C03654=1204.977,411.495,-82.961,-175.836,8.473,148.470
C03655=1204.981,411.248,-82.925,-175.837,8.471,148.469
C03656=1204.985,411.000,-82.891,-175.837,8.469,148.469
C03657=1204.989,410.753,-82.855,-175.837,8.467,148.468
C03658=1204.993,410.506,-82.820,-175.838,8.464,148.468
C03659=1204.997,410.258,-82.785,-175.838,8.462,148.467
C03660=1205.001,410.011,-82.749,-175.839,8.460,148.467
C03661=1205.005,409.764,-82.714,-175.839,8.458,148.466
C03662=1205.009,409.516,-82.679,-175.839,8.456,148.466
C03663=1205.013,409.268,-82.644,-175.839,8.453,148.465
C03664=1205.017,409.021,-82.609,-175.840,8.451,148.465
C03665=1205.021,408.773,-82.574,-175.840,8.449,148.464
C03666=1205.025,408.525,-82.539,-175.840,8.447,148.464
C03667=1205.029,408.278,-82.504,-175.840,8.445,148.463
C03668=1205.032,408.031,-82.469,-175.841,8.443,148.463
C03669=1205.037,407.784,-82.434,-175.841,8.440,148.462
C03670=1205.040,407.536,-82.399,-175.842,8.438,148.462
C03671=1205.044,407.288,-82.364,-175.842,8.436,148.461
C03672=1205.049,407.041,-82.329,-175.842,8.433,148.461
C03673=1205.053,406.793,-82.294,-175.843,8.431,148.460
C03674=1205.057,406.546,-82.259,-175.843,8.428,148.460
C03675=1205.061,406.298,-82.224,-175.844,8.426,148.459
C03676=1205.065,406.051,-82.188,-175.844,8.424,148.459
C03677=1205.069,405.803,-82.154,-175.844,8.422,148.458
C03678=1205.073,405.556,-82.118,-175.845,8.420,148.458
C03679=1205.077,405.308,-82.084,-175.845,8.417,148.457
C03680=1205.081,405.061,-82.048,-175.845,8.415,148.457
C03681=1205.085,404.813,-82.014,-175.846,8.412,148.456
C03682=1205.089,404.566,-81.978,-175.847,8.410,148.456
C03683=1205.093,404.318,-81.944,-175.847,8.408,148.455
C03684=1205.098,404.071,-81.908,-175.847,8.405,148.455
C03685=1205.101,403.823,-81.874,-175.847,8.403,148.454
C03686=1205.104,403.576,-81.839,-175.848,8.401,148.454
C03687=1205.109,403.328,-81.804,-175.849,8.398,148.453
C03688=1205.113,403.081,-81.769,-175.849,8.396,148.453
C03689=1205.117,402.833,-81.734,-175.849,8.394,148.452
C03690=1205.121,402.586,-81.699,-175.849,8.391,148.452
C03691=1205.125,402.338,-81.664,-175.850,8.389,148.451
C03692=1205.129,402.090,-81.629,-175.851,8.386,148.451
C03693=1205.133,401.843,-81.594,-175.851,8.384,148.450
C03694=1205.138,401.595,-81.559,-175.851,8.382,148.450
C03695=1205.141,401.348,-81.524,-175.852,8.379,148.449
C03696=1205.145,401.101,-81.490,-175.852,8.376,148.449
C03697=1205.149,400.853,-81.455,-175.853,8.374,148.448
C03698=1205.153,400.606,-81.420,-175.853,8.372,148.448
C03699=1205.157,400.358,-81.385,-175.853,8.370,148.447
C03700=1205.162,400.111,-81.350,-175.854,8.367,148.447
C03701=1205.166,399.863,-81.315,-175.854,8.364,148.446
C03702=1205.170,399.615,-81.280,-175.855,8.362,148.446
C03703=1205.173,399.368,-81.246,-175.856,8.359,148.445
C03704=1205.177,399.120,-81.211,-175.856,8.357,148.445
C03705=1205.182,398.873,-81.176,-175.856,8.355,148.444
C03706=1205.185,398.625,-81.141,-175.857,8.352,148.444
C03707=1205.190,398.378,-81.106,-175.858,8.350,148.443
C03708=1205.194,398.130,-81.071,-175.858,8.347,148.443
C03709=1205.197,397.883,-81.037,-175.859,8.344,148.442
C03710=1205.201,397.635,-81.002,-175.859,8.342,148.442
C03711=1205.206,397.388,-80.968,-175.860,8.340,148.441
C03712=1205.210,397.140,-80.932,-175.860,8.337,148.441
C03713=1205.214,396.893,-80.898,-175.861,8.335,148.440
C03714=1205.218,396.645,-80.863,-175.861,8.332,148.440
C03715=1205.222,396.398,-80.828,-175.862,8.329,148.439
C03716=1205.226,396.150,-80.793,-175.862,8.327,148.439
C03717=1205.230,395.903,-80.759,-175.863,8.324,148.438
C03718=1205.234,395.654,-80.724,-175.863,8.322,148.438
C03719=1205.238,395.408,-80.689,-175.864,8.319,148.437
C03720=1205.242,395.160,-80.655,-175.865,8.317,148.437
C03721=1205.246,394.912,-80.620,-175.865,8.314,148.436
C03722=1205.250,394.664,-80.585,-175.866,8.312,148.436
C03723=1205.254,394.417,-80.550,-175.866,8.309,148.435
C03724=1205.258,394.170,-80.516,-175.867,8.307,148.435
C03725=1205.262,393.922,-80.481,-175.868,8.303,148.434
C03726=1205.266,393.674,-80.447,-175.868,8.301,148.433
C03727=1205.270,393.427,-80.411,-175.869,8.298,148.433
C03728=1205.274,393.180,-80.377,-175.869,8.296,148.433
C03729=1205.279,392.896,-80.337,-175.870,8.293,148.432
C03730=1205.283,392.614,-80.298,-175.871,8.290,148.431
C03731=1205.288,392.332,-80.259,-175.872,8.287,148.431
C03732=1205.293,392.049,-80.219,-175.873,8.284,148.430
C03733=1205.297,391.801,-80.184,-175.873,8.281,148.430
C03734=1205.301,391.554,-80.150,-175.873,8.278,148.429
C03735=1205.305,391.306,-80.115,-175.874,8.276,148.429
C03736=1205.309,391.059,-80.080,-175.875,8.273,148.428
C03737=1205.312,390.811,-80.046,-175.876,8.270,148.428
C03738=1205.317,390.564,-80.012,-175.876,8.268,148.427
C03739=1205.321,390.316,-79.977,-175.877,8.265,148.427
C03740=1205.325,390.068,-79.942,-175.877,8.263,148.426
C03741=1205.328,389.821,-79.908,-175.879,8.260,148.426
C03742=1205.333,389.573,-79.874,-175.879,8.257,148.425
C03743=1205.337,389.326,-79.839,-175.880,8.255,148.425
C03744=1205.341,389.078,-79.805,-175.881,8.252,148.424
C03745=1205.345,388.830,-79.770,-175.881,8.249,148.424
C03746=1205.349,388.583,-79.735,-175.882,8.246,148.423
C03747=1205.353,388.336,-79.701,-175.883,8.244,148.423
C03748=1205.357,388.088,-79.666,-175.884,8.240,148.422
C03749=1205.361,387.840,-79.632,-175.884,8.238,148.422
C03750=1205.365,387.593,-79.598,-175.885,8.235,148.421
C03751=1205.369,387.345,-79.563,-175.886,8.232,148.421
C03752=1205.374,387.098,-79.529,-175.887,8.229,148.420
C03753=1205.377,386.850,-79.494,-175.887,8.227,148.420
C03754=1205.381,386.602,-79.460,-175.888,8.224,148.419
C03755=1205.385,386.355,-79.426,-175.889,8.221,148.419
C03756=1205.389,386.107,-79.391,-175.890,8.218,148.418
C03757=1205.394,385.860,-79.357,-175.891,8.215,148.418
C03758=1205.397,385.612,-79.322,-175.891,8.213,148.417
C03759=1205.402,385.365,-79.288,-175.893,8.210,148.417
C03760=1205.406,385.116,-79.253,-175.893,8.207,148.416
C03761=1205.409,384.869,-79.219,-175.894,8.204,148.416
C03762=1205.414,384.622,-79.185,-175.895,8.201,148.415
C03763=1205.417,384.374,-79.151,-175.896,8.199,148.415
C03764=1205.422,384.127,-79.116,-175.897,8.196,148.414
C03765=1205.425,383.879,-79.082,-175.898,8.193,148.414
C03766=1205.430,383.631,-79.048,-175.899,8.190,148.413
C03767=1205.434,383.383,-79.014,-175.900,8.187,148.413
C03768=1205.438,383.136,-78.979,-175.901,8.184,148.412
C03769=1205.442,382.888,-78.945,-175.902,8.181,148.412
C03770=1205.446,382.641,-78.911,-175.903,8.178,148.411
C03771=1205.450,382.393,-78.876,-175.903,8.176,148.411
C03772=1205.454,382.146,-78.842,-175.904,8.173,148.410
C03773=1205.458,381.898,-78.808,-175.905,8.171,148.410
C03774=1205.462,381.650,-78.774,-175.906,8.167,148.409
C03775=1205.467,381.403,-78.740,-175.907,8.165,148.409
C03776=1205.471,381.154,-78.705,-175.908,8.162,148.408
C03777=1205.474,380.907,-78.671,-175.909,8.159,148.408
C03778=1205.479,380.660,-78.637,-175.911,8.156,148.408
C03779=1205.482,380.412,-78.603,-175.911,8.153,148.407
C03780=1205.487,380.164,-78.569,-175.913,8.150,148.407
C03781=1205.491,379.917,-78.535,-175.913,8.147,148.406
C03782=1205.495,379.669,-78.500,-175.915,8.144,148.406
C03783=1205.499,379.422,-78.466,-175.916,8.141,148.405
C03784=1205.503,379.174,-78.432,-175.916,8.138,148.405
C03785=1205.507,378.926,-78.398,-175.918,8.135,148.404
C03786=1205.511,378.678,-78.364,-175.919,8.133,148.404
C03787=1205.515,378.431,-78.330,-175.920,8.129,148.403
C03788=1205.518,378.184,-78.296,-175.921,8.127,148.403
C03789=1205.523,377.936,-78.262,-175.922,8.124,148.402
C03790=1205.527,377.688,-78.228,-175.923,8.121,148.402
C03791=1205.532,377.441,-78.194,-175.924,8.118,148.401
C03792=1205.535,377.193,-78.160,-175.926,8.114,148.401
C03793=1205.540,376.945,-78.126,-175.927,8.111,148.401
C03794=1205.544,376.698,-78.092,-175.928,8.108,148.400
C03795=1205.547,376.450,-78.058,-175.929,8.106,148.400
C03796=1205.552,376.202,-78.024,-175.930,8.103,148.399
C03797=1205.556,375.955,-77.990,-175.931,8.100,148.399
C03798=1205.560,375.707,-77.956,-175.933,8.097,148.398
C03799=1205.564,375.459,-77.922,-175.933,8.094,148.398
C03800=1205.568,375.212,-77.888,-175.935,8.090,148.397
C03801=1205.572,374.964,-77.854,-175.936,8.088,148.397
C03802=1205.576,374.716,-77.820,-175.938,8.085,148.397
C03803=1205.581,374.468,-77.786,-175.939,8.082,148.396
C03804=1205.584,374.221,-77.752,-175.940,8.079,148.396
C03805=1205.588,373.974,-77.718,-175.941,8.076,148.396
C03806=1205.592,373.725,-77.684,-175.943,8.072,148.395
C03807=1205.596,373.478,-77.650,-175.944,8.070,148.394
C03808=1205.600,373.230,-77.617,-175.945,8.067,148.394
C03809=1205.605,372.983,-77.583,-175.946,8.064,148.394
C03810=1205.609,372.735,-77.549,-175.947,8.061,148.393
C03811=1205.612,372.487,-77.515,-175.949,8.058,148.393
C03812=1205.617,372.239,-77.482,-175.950,8.055,148.392
C03813=1205.621,371.992,-77.448,-175.952,8.052,148.392
C03814=1205.625,371.744,-77.414,-175.953,8.049,148.392
C03815=1205.629,371.496,-77.380,-175.955,8.045,148.391
C03816=1205.633,371.249,-77.347,-175.956,8.043,148.391
C03817=1205.637,371.002,-77.313,-175.957,8.040,148.390
C03818=1205.641,370.754,-77.280,-175.958,8.037,148.390
C03819=1205.645,370.506,-77.245,-175.960,8.033,148.390
C03820=1205.649,370.258,-77.212,-175.961,8.031,148.389
C03821=1205.653,370.011,-77.178,-175.962,8.028,148.389
C03822=1205.657,369.763,-77.145,-175.964,8.024,148.388
C03823=1205.662,369.515,-77.111,-175.965,8.021,148.388
C03824=1205.665,369.267,-77.077,-175.966,8.019,148.388
C03825=1205.670,369.020,-77.044,-175.968,8.015,148.387
C03826=1205.673,368.773,-77.010,-175.970,8.012,148.387
C03827=1205.678,368.524,-76.976,-175.971,8.010,148.387
C03828=1205.682,368.277,-76.943,-175.973,8.006,148.386
C03829=1205.686,368.030,-76.909,-175.974,8.003,148.386
C03830=1205.690,367.781,-76.875,-175.975,8.000,148.385
C03831=1205.695,367.533,-76.842,-175.977,7.997,148.385
C03832=1205.699,367.286,-76.808,-175.978,7.994,148.385
C03833=1205.703,367.005,-76.771,-175.980,7.990,148.384
C03834=1205.708,366.725,-76.732,-175.982,7.987,148.384
C03835=1205.712,366.445,-76.695,-175.983,7.984,148.383
C03836=1205.717,366.164,-76.656,-175.985,7.980,148.383
C03837=1205.721,365.917,-76.623,-175.987,7.977,148.383
C03838=1205.725,365.669,-76.590,-175.988,7.974,148.382
C03839=1205.729,365.421,-76.557,-175.990,7.971,148.382
C03840=1205.733,365.173,-76.522,-175.992,7.968,148.382
C03841=1205.737,364.925,-76.489,-175.993,7.965,148.381
C03842=1205.742,364.678,-76.455,-175.995,7.961,148.381
C03843=1205.746,364.430,-76.422,-175.996,7.959,148.381
C03844=1205.750,364.182,-76.389,-175.998,7.955,148.380
C03845=1205.754,363.935,-76.355,-175.999,7.952,148.380
C03846=1205.758,363.687,-76.322,-176.001,7.949,148.380
C03847=1205.762,363.440,-76.289,-176.003,7.946,148.379
C03848=1205.766,363.191,-76.255,-176.004,7.944,148.379
C03849=1205.770,362.943,-76.222,-176.006,7.940,148.379
C03850=1205.774,362.696,-76.189,-176.007,7.937,148.378
C03851=1205.778,362.448,-76.156,-176.009,7.934,148.378
C03852=1205.782,362.200,-76.123,-176.011,7.931,148.378
C03853=1205.787,361.953,-76.088,-176.012,7.927,148.377
C03854=1205.791,361.705,-76.055,-176.014,7.925,148.377
C03855=1205.795,361.457,-76.022,-176.016,7.921,148.376
C03856=1205.799,361.210,-75.989,-176.018,7.919,148.376
C03857=1205.803,360.962,-75.956,-176.019,7.915,148.376
C03858=1205.807,360.714,-75.923,-176.021,7.913,148.376
C03859=1205.811,360.466,-75.889,-176.023,7.909,148.375
C03860=1205.816,360.219,-75.856,-176.024,7.906,148.375
C03861=1205.820,359.971,-75.823,-176.026,7.903,148.375
C03862=1205.823,359.723,-75.790,-176.028,7.900,148.374
C03863=1205.827,359.475,-75.756,-176.030,7.897,148.374
C03864=1205.832,359.227,-75.723,-176.031,7.894,148.374
C03865=1205.836,358.979,-75.690,-176.033,7.891,148.373
C03866=1205.839,358.732,-75.658,-176.035,7.888,148.373
C03867=1205.843,358.484,-75.624,-176.036,7.884,148.373
C03868=1205.847,358.236,-75.591,-176.038,7.882,148.373
C03869=1205.852,357.989,-75.558,-176.040,7.879,148.372
C03870=1205.856,357.740,-75.526,-176.042,7.875,148.372
C03871=1205.860,357.493,-75.492,-176.044,7.872,148.372
C03872=1205.864,357.245,-75.459,-176.046,7.869,148.371
C03873=1205.868,356.997,-75.426,-176.047,7.866,148.371
C03874=1205.873,356.749,-75.393,-176.049,7.863,148.371
C03875=1205.877,356.502,-75.360,-176.050,7.860,148.370
C03876=1205.881,356.254,-75.327,-176.053,7.857,148.370
C03877=1205.885,356.006,-75.294,-176.054,7.854,148.370
C03878=1205.889,355.758,-75.262,-176.056,7.851,148.370
C03879=1205.893,355.510,-75.229,-176.058,7.848,148.369
C03880=1205.897,355.263,-75.195,-176.060,7.845,148.369
C03881=1205.901,355.015,-75.162,-176.062,7.841,148.369
C03882=1205.906,354.767,-75.130,-176.063,7.839,148.369
C03883=1205.910,354.520,-75.097,-176.066,7.835,148.368
C03884=1205.914,354.272,-75.064,-176.067,7.833,148.368
C03885=1205.918,354.025,-75.031,-176.069,7.829,148.368
C03886=1205.922,353.776,-74.999,-176.071,7.827,148.368
C03887=1205.926,353.528,-74.966,-176.073,7.823,148.367
C03888=1205.930,353.281,-74.933,-176.075,7.820,148.367
C03889=1205.935,353.033,-74.899,-176.076,7.817,148.367
C03890=1205.938,352.785,-74.868,-176.079,7.814,148.366
C03891=1205.942,352.537,-74.834,-176.080,7.811,148.366
C03892=1205.947,352.289,-74.801,-176.082,7.808,148.366
C03893=1205.951,352.041,-74.769,-176.084,7.805,148.366
C03894=1205.955,351.793,-74.736,-176.086,7.802,148.365
C03895=1205.959,351.545,-74.704,-176.088,7.798,148.365
C03896=1205.964,351.298,-74.671,-176.090,7.796,148.365
C03897=1205.968,351.051,-74.638,-176.092,7.792,148.365
C03898=1205.972,350.802,-74.605,-176.094,7.790,148.365
C03899=1205.976,350.555,-74.573,-176.096,7.787,148.364
C03900=1205.980,350.306,-74.540,-176.097,7.784,148.364
C03901=1205.984,350.059,-74.507,-176.099,7.780,148.364
C03902=1205.988,349.811,-74.475,-176.101,7.777,148.364
C03903=1205.992,349.563,-74.442,-176.103,7.775,148.363
C03904=1205.997,349.315,-74.410,-176.105,7.771,148.363
C03905=1206.001,349.068,-74.377,-176.107,7.769,148.363
C03906=1206.005,348.820,-74.345,-176.109,7.765,148.363
C03907=1206.009,348.572,-74.312,-176.111,7.762,148.363
C03908=1206.014,348.323,-74.280,-176.113,7.760,148.362
C03909=1206.017,348.076,-74.247,-176.115,7.756,148.362
C03910=1206.022,347.828,-74.215,-176.117,7.754,148.362
C03911=1206.026,347.581,-74.182,-176.119,7.750,148.362
C03912=1206.030,347.333,-74.150,-176.121,7.747,148.362
C03913=1206.034,347.085,-74.117,-176.123,7.745,148.361
C03914=1206.038,346.837,-74.085,-176.125,7.741,148.361
C03915=1206.042,346.589,-74.052,-176.127,7.739,148.361
C03916=1206.047,346.342,-74.020,-176.129,7.735,148.361
C03917=1206.051,346.093,-73.988,-176.131,7.732,148.360
C03918=1206.055,345.846,-73.955,-176.133,7.729,148.360
C03919=1206.058,345.598,-73.923,-176.135,7.726,148.360
C03920=1206.063,345.349,-73.890,-176.137,7.724,148.360
C03921=1206.068,345.102,-73.858,-176.139,7.720,148.360
C03922=1206.071,344.854,-73.826,-176.141,7.717,148.359
C03923=1206.076,344.606,-73.793,-176.143,7.714,148.359
C03924=1206.079,344.358,-73.761,-176.145,7.711,148.359
C03925=1206.084,344.111,-73.729,-176.147,7.709,148.359
C03926=1206.088,343.863,-73.697,-176.149,7.705,148.359
C03927=1206.092,343.614,-73.664,-176.151,7.702,148.358
C03928=1206.096,343.366,-73.633,-176.153,7.699,148.358
C03929=1206.101,343.119,-73.600,-176.155,7.696,148.358
C03930=1206.104,342.871,-73.568,-176.157,7.694,148.358
C03931=1206.109,342.623,-73.535,-176.159,7.690,148.358
C03932=1206.113,342.375,-73.504,-176.162,7.687,148.358
C03933=1206.118,342.127,-73.472,-176.163,7.685,148.357
C03934=1206.121,341.880,-73.439,-176.166,7.681,148.357
C03935=1206.125,341.632,-73.407,-176.167,7.679,148.357
C03936=1206.129,341.384,-73.375,-176.169,7.675,148.357
C03937=1206.134,341.106,-73.338,-176.172,7.672,148.357
C03938=1206.140,340.827,-73.303,-176.174,7.669,148.357
C03939=1206.144,340.549,-73.266,-176.177,7.666,148.356
C03940=1206.148,340.271,-73.231,-176.179,7.662,148.356
C03941=1206.153,340.023,-73.198,-176.181,7.659,148.356
C03942=1206.157,339.775,-73.167,-176.183,7.657,148.356
C03943=1206.162,339.527,-73.134,-176.185,7.653,148.356
C03944=1206.165,339.279,-73.103,-176.188,7.650,148.356
C03945=1206.169,339.031,-73.071,-176.189,7.648,148.355
C03946=1206.174,338.783,-73.039,-176.191,7.644,148.355
C03947=1206.178,338.535,-73.007,-176.194,7.641,148.355
C03948=1206.181,338.287,-72.975,-176.196,7.639,148.355
C03949=1206.187,338.040,-72.943,-176.198,7.635,148.355
C03950=1206.190,337.792,-72.911,-176.200,7.633,148.355
C03951=1206.194,337.544,-72.879,-176.202,7.630,148.354
C03952=1206.199,337.296,-72.847,-176.204,7.627,148.354
C03953=1206.203,337.048,-72.815,-176.206,7.624,148.354
C03954=1206.206,336.800,-72.783,-176.208,7.621,148.354
C03955=1206.211,336.552,-72.751,-176.211,7.618,148.354
C03956=1206.215,336.304,-72.720,-176.213,7.615,148.354
C03957=1206.219,336.057,-72.688,-176.215,7.612,148.354
C03958=1206.224,335.808,-72.656,-176.217,7.609,148.353
C03959=1206.228,335.560,-72.625,-176.219,7.606,148.353
C03960=1206.232,335.312,-72.593,-176.221,7.603,148.353
C03961=1206.236,335.064,-72.561,-176.223,7.600,148.353
C03962=1206.240,334.816,-72.529,-176.226,7.597,148.353
C03963=1206.245,334.569,-72.497,-176.228,7.594,148.353
C03964=1206.248,334.321,-72.465,-176.230,7.591,148.353
C03965=1206.253,334.073,-72.435,-176.232,7.588,148.353
C03966=1206.257,333.824,-72.402,-176.234,7.586,148.352
C03967=1206.261,333.576,-72.370,-176.236,7.583,148.352
C03968=1206.265,333.329,-72.339,-176.239,7.580,148.352
C03969=1206.269,333.081,-72.307,-176.241,7.577,148.352
C03970=1206.274,332.833,-72.276,-176.243,7.574,148.352
C03971=1206.278,332.585,-72.244,-176.245,7.571,148.352
C03972=1206.283,332.337,-72.212,-176.247,7.568,148.352
C03973=1206.287,332.089,-72.181,-176.250,7.565,148.352
C03974=1206.291,331.841,-72.150,-176.251,7.563,148.351
C03975=1206.295,331.593,-72.118,-176.254,7.560,148.351
C03976=1206.299,331.344,-72.086,-176.256,7.556,148.351
C03977=1206.304,331.097,-72.055,-176.258,7.554,148.351
C03978=1206.307,330.849,-72.023,-176.261,7.551,148.351
C03979=1206.312,330.601,-71.992,-176.263,7.547,148.351
C03980=1206.316,330.353,-71.960,-176.265,7.545,148.351
C03981=1206.320,330.106,-71.929,-176.267,7.542,148.351
C03982=1206.324,329.857,-71.898,-176.269,7.540,148.351
C03983=1206.328,329.610,-71.866,-176.272,7.536,148.350
C03984=1206.332,329.361,-71.835,-176.274,7.533,148.350
C03985=1206.337,329.113,-71.803,-176.276,7.531,148.350
C03986=1206.341,328.865,-71.772,-176.279,7.528,148.350
C03987=1206.346,328.617,-71.740,-176.281,7.524,148.350
C03988=1206.349,328.369,-71.709,-176.283,7.522,148.350
C03989=1206.354,328.121,-71.678,-176.285,7.519,148.350
C03990=1206.358,327.873,-71.646,-176.287,7.517,148.350
C03991=1206.362,327.625,-71.615,-176.289,7.513,148.350
C03992=1206.366,327.377,-71.583,-176.292,7.510,148.350
C03993=1206.371,327.129,-71.553,-176.294,7.508,148.350
C03994=1206.375,326.881,-71.522,-176.296,7.505,148.350
C03995=1206.379,326.633,-71.490,-176.299,7.501,148.349
C03996=1206.384,326.385,-71.459,-176.301,7.499,148.349
C03997=1206.387,326.137,-71.427,-176.303,7.496,148.349
C03998=1206.392,325.889,-71.397,-176.305,7.494,148.349
C03999=1206.396,325.641,-71.365,-176.307,7.490,148.349
C04000=1206.400,325.393,-71.334,-176.310,7.487,148.349
C04001=1206.404,325.145,-71.303,-176.312,7.485,148.349
C04002=1206.408,324.897,-71.271,-176.314,7.482,148.349
C04003=1206.413,324.649,-71.241,-176.317,7.479,148.349
C04004=1206.417,324.401,-71.209,-176.319,7.476,148.349
C04005=1206.421,324.153,-71.178,-176.321,7.473,148.349
C04006=1206.425,323.905,-71.147,-176.323,7.471,148.348
C04007=1206.429,323.657,-71.117,-176.326,7.468,148.348
C04008=1206.433,323.409,-71.085,-176.328,7.464,148.348
C04009=1206.438,323.161,-71.054,-176.330,7.462,148.348
C04010=1206.442,322.913,-71.023,-176.333,7.459,148.348
C04011=1206.446,322.664,-70.992,-176.335,7.456,148.348
C04012=1206.451,322.417,-70.961,-176.337,7.453,148.348
C04013=1206.455,322.169,-70.930,-176.340,7.450,148.348
C04014=1206.458,321.921,-70.899,-176.341,7.448,148.348
C04015=1206.463,321.673,-70.869,-176.344,7.445,148.348
C04016=1206.467,321.424,-70.837,-176.347,7.442,148.348
C04017=1206.471,321.177,-70.806,-176.348,7.439,148.348
C04018=1206.476,320.929,-70.775,-176.351,7.436,148.348
C04019=1206.480,320.680,-70.744,-176.353,7.434,148.348
C04020=1206.484,320.433,-70.714,-176.355,7.431,148.348
C04021=1206.488,320.185,-70.683,-176.358,7.428,148.348
C04022=1206.492,319.936,-70.652,-176.360,7.425,148.348
C04023=1206.497,319.688,-70.621,-176.362,7.422,148.347
C04024=1206.502,319.440,-70.591,-176.365,7.419,148.347
C04025=1206.505,319.192,-70.559,-176.367,7.417,148.348
C04026=1206.509,318.944,-70.528,-176.369,7.414,148.347
C04027=1206.514,318.696,-70.498,-176.372,7.411,148.347
C04028=1206.518,318.448,-70.467,-176.374,7.408,148.347
C04029=1206.522,318.200,-70.436,-176.376,7.405,148.347
C04030=1206.526,317.952,-70.406,-176.379,7.403,148.347
C04031=1206.531,317.704,-70.375,-176.381,7.400,148.347
C04032=1206.534,317.456,-70.344,-176.383,7.398,148.347
C04033=1206.539,317.208,-70.314,-176.386,7.394,148.347
C04034=1206.544,316.960,-70.283,-176.388,7.391,148.347
C04035=1206.548,316.711,-70.252,-176.390,7.389,148.347
C04036=1206.551,316.464,-70.222,-176.393,7.386,148.347
C04037=1206.556,316.216,-70.191,-176.395,7.383,148.347
C04038=1206.561,315.967,-70.161,-176.397,7.380,148.347
C04039=1206.564,315.719,-70.130,-176.400,7.377,148.347
C04040=1206.569,315.471,-70.099,-176.402,7.375,148.347
C04041=1206.574,315.195,-70.065,-176.405,7.372,148.347
C04042=1206.579,314.919,-70.032,-176.407,7.369,148.347
C04043=1206.583,314.643,-69.997,-176.410,7.366,148.347
C04044=1206.588,314.367,-69.963,-176.413,7.363,148.347
C04045=1206.592,314.118,-69.933,-176.415,7.360,148.347
C04046=1206.596,313.870,-69.902,-176.418,7.357,148.347
C04047=1206.600,313.622,-69.872,-176.420,7.354,148.347
C04048=1206.605,313.375,-69.842,-176.422,7.351,148.347
C04049=1206.609,313.126,-69.810,-176.424,7.349,148.347
C04050=1206.613,312.878,-69.781,-176.427,7.346,148.347
C04051=1206.618,312.630,-69.750,-176.430,7.343,148.347
C04052=1206.622,312.382,-69.720,-176.432,7.341,148.347
C04053=1206.626,312.134,-69.689,-176.434,7.337,148.347
C04054=1206.630,311.886,-69.660,-176.436,7.335,148.347
C04055=1206.634,311.637,-69.629,-176.439,7.332,148.347
C04056=1206.638,311.389,-69.598,-176.442,7.329,148.347
C04057=1206.643,311.141,-69.568,-176.444,7.327,148.347
C04058=1206.647,310.893,-69.538,-176.446,7.324,148.347
C04059=1206.652,310.645,-69.508,-176.448,7.321,148.347
C04060=1206.656,310.397,-69.478,-176.451,7.318,148.347
C04061=1206.660,310.148,-69.447,-176.453,7.315,148.347
C04062=1206.664,309.901,-69.417,-176.456,7.313,148.347
C04063=1206.669,309.652,-69.387,-176.458,7.310,148.347
C04064=1206.673,309.404,-69.357,-176.460,7.308,148.347
C04065=1206.677,309.156,-69.326,-176.463,7.305,148.347
C04066=1206.681,308.908,-69.296,-176.466,7.302,148.347
C04067=1206.686,308.660,-69.266,-176.467,7.299,148.347
C04068=1206.690,308.412,-69.236,-176.470,7.296,148.347
C04069=1206.695,308.164,-69.205,-176.472,7.294,148.347
C04070=1206.698,307.915,-69.176,-176.475,7.291,148.347
C04071=1206.702,307.667,-69.145,-176.477,7.289,148.347
C04072=1206.707,307.419,-69.115,-176.480,7.286,148.347
C04073=1206.711,307.171,-69.085,-176.482,7.283,148.347
C04074=1206.716,306.923,-69.055,-176.484,7.281,148.347
C04075=1206.720,306.675,-69.025,-176.487,7.278,148.347
C04076=1206.724,306.427,-68.995,-176.489,7.275,148.347
C04077=1206.729,306.178,-68.965,-176.492,7.272,148.347
C04078=1206.733,305.930,-68.935,-176.494,7.269,148.347
C04079=1206.737,305.682,-68.906,-176.496,7.267,148.347
C04080=1206.742,305.434,-68.875,-176.499,7.264,148.347
C04081=1206.746,305.186,-68.846,-176.501,7.262,148.347
C04082=1206.751,304.937,-68.816,-176.504,7.258,148.347
C04083=1206.755,304.690,-68.785,-176.506,7.256,148.347
C04084=1206.759,304.442,-68.756,-176.509,7.253,148.347
C04085=1206.763,304.193,-68.726,-176.511,7.250,148.347
C04086=1206.768,303.945,-68.696,-176.513,7.248,148.347
C04087=1206.772,303.697,-68.666,-176.516,7.245,148.347
C04088=1206.775,303.448,-68.636,-176.518,7.243,148.347
C04089=1206.780,303.200,-68.606,-176.521,7.240,148.347
C04090=1206.784,302.952,-68.576,-176.523,7.238,148.347
C04091=1206.788,302.704,-68.547,-176.526,7.235,148.347
C04092=1206.792,302.455,-68.517,-176.528,7.232,148.347
C04093=1206.797,302.207,-68.487,-176.531,7.229,148.347
C04094=1206.802,301.960,-68.457,-176.533,7.226,148.347
C04095=1206.806,301.712,-68.428,-176.535,7.224,148.347
C04096=1206.810,301.463,-68.399,-176.538,7.221,148.347
C04097=1206.815,301.215,-68.368,-176.540,7.219,148.347
C04098=1206.819,300.967,-68.338,-176.543,7.216,148.347
C04099=1206.823,300.719,-68.309,-176.545,7.214,148.347
C04100=1206.827,300.470,-68.279,-176.548,7.211,148.347
C04101=1206.832,300.222,-68.250,-176.550,7.208,148.347
C04102=1206.836,299.974,-68.221,-176.552,7.205,148.347
C04103=1206.841,299.725,-68.190,-176.555,7.202,148.347
C04104=1206.845,299.478,-68.160,-176.557,7.200,148.348
C04105=1206.849,299.229,-68.131,-176.560,7.197,148.348
C04106=1206.853,298.981,-68.101,-176.562,7.195,148.348
C04107=1206.857,298.733,-68.072,-176.565,7.192,148.348
C04108=1206.861,298.485,-68.042,-176.567,7.190,148.348
C04109=1206.865,298.236,-68.013,-176.570,7.187,148.348
C04110=1206.870,297.988,-67.984,-176.572,7.185,148.348
C04111=1206.875,297.740,-67.954,-176.574,7.182,148.348
C04112=1206.879,297.492,-67.924,-176.578,7.179,148.348
C04113=1206.884,297.244,-67.895,-176.580,7.177,148.348
C04114=1206.888,296.995,-67.866,-176.582,7.174,148.348
C04115=1206.892,296.747,-67.836,-176.585,7.171,148.348
C04116=1206.896,296.499,-67.807,-176.587,7.168,148.348
C04117=1206.900,296.251,-67.777,-176.589,7.166,148.348
C04118=1206.904,296.002,-67.748,-176.592,7.163,148.348
C04119=1206.909,295.754,-67.718,-176.594,7.161,148.348
C04120=1206.913,295.506,-67.689,-176.597,7.158,148.348
C04121=1206.918,295.258,-67.660,-176.599,7.156,148.348
C04122=1206.922,295.009,-67.631,-176.602,7.153,148.348
C04123=1206.926,294.761,-67.602,-176.604,7.150,148.348
C04124=1206.930,294.513,-67.572,-176.607,7.148,148.349
C04125=1206.935,294.265,-67.543,-176.610,7.145,148.349
C04126=1206.939,294.016,-67.513,-176.612,7.143,148.349
C04127=1206.943,293.768,-67.484,-176.614,7.140,148.349
C04128=1206.948,293.520,-67.455,-176.617,7.137,148.349
C04129=1206.952,293.272,-67.426,-176.619,7.134,148.349
C04130=1206.956,293.023,-67.396,-176.621,7.132,148.349
C04131=1206.961,292.775,-67.367,-176.624,7.129,148.349
C04132=1206.965,292.527,-67.338,-176.626,7.127,148.349
C04133=1206.970,292.279,-67.309,-176.629,7.124,148.349
C04134=1206.973,292.031,-67.280,-176.632,7.122,148.349
C04135=1206.977,291.782,-67.251,-176.634,7.119,148.349
C04136=1206.982,291.534,-67.221,-176.636,7.117,148.349
C04137=1206.986,291.285,-67.193,-176.639,7.114,148.349
C04138=1206.991,291.038,-67.164,-176.641,7.112,148.350
C04139=1206.995,290.789,-67.134,-176.644,7.109,148.350
C04140=1207.000,290.540,-67.105,-176.646,7.107,148.350
C04141=1207.004,290.292,-67.076,-176.649,7.104,148.350
C04142=1207.008,290.045,-67.047,-176.651,7.101,148.350
C04143=1207.012,289.796,-67.019,-176.654,7.098,148.350
C04144=1207.017,289.548,-66.989,-176.656,7.096,148.350
C04145=1207.021,289.273,-66.958,-176.659,7.094,148.350
C04146=1207.027,288.999,-66.925,-176.662,7.090,148.350
C04147=1207.031,288.725,-66.893,-176.665,7.087,148.350
C04148=1207.036,288.451,-66.861,-176.668,7.085,148.351
C04149=1207.040,288.202,-66.832,-176.670,7.083,148.351
C04150=1207.044,287.954,-66.804,-176.673,7.080,148.351
C04151=1207.048,287.706,-66.774,-176.675,7.077,148.351
C04152=1207.053,287.457,-66.746,-176.677,7.074,148.351
C04153=1207.058,287.209,-66.716,-176.680,7.072,148.351
C04154=1207.061,286.961,-66.688,-176.683,7.069,148.351
C04155=1207.066,286.713,-66.659,-176.685,7.067,148.351
C04156=1207.071,286.464,-66.631,-176.688,7.064,148.351
C04157=1207.075,286.216,-66.601,-176.690,7.062,148.351
C04158=1207.079,285.968,-66.573,-176.693,7.059,148.351
C04159=1207.083,285.720,-66.544,-176.695,7.057,148.352
C04160=1207.088,285.471,-66.515,-176.697,7.055,148.352
C04161=1207.093,285.223,-66.487,-176.700,7.052,148.352
C04162=1207.096,284.975,-66.458,-176.702,7.050,148.352
C04163=1207.101,284.726,-66.429,-176.705,7.047,148.352
C04164=1207.106,284.478,-66.400,-176.707,7.045,148.352
C04165=1207.109,284.230,-66.372,-176.710,7.042,148.352
C04166=1207.114,283.981,-66.343,-176.712,7.040,148.352
C04167=1207.119,283.733,-66.314,-176.715,7.037,148.352
C04168=1207.122,283.485,-66.286,-176.717,7.035,148.352
C04169=1207.127,283.236,-66.257,-176.720,7.032,148.352
C04170=1207.132,282.988,-66.228,-176.722,7.029,148.353
C04171=1207.135,282.740,-66.200,-176.725,7.027,148.353
C04172=1207.140,282.491,-66.172,-176.727,7.025,148.353
C04173=1207.144,282.243,-66.143,-176.730,7.022,148.353
C04174=1207.148,281.995,-66.114,-176.732,7.019,148.353
C04175=1207.153,281.746,-66.086,-176.735,7.018,148.353
C04176=1207.157,281.498,-66.057,-176.738,7.014,148.353
C04177=1207.162,281.250,-66.029,-176.740,7.012,148.353
C04178=1207.166,281.002,-66.000,-176.742,7.009,148.353
C04179=1207.170,280.753,-65.972,-176.745,7.007,148.354
C04180=1207.175,280.505,-65.944,-176.748,7.004,148.354
C04181=1207.179,280.256,-65.915,-176.750,7.002,148.354
C04182=1207.183,280.008,-65.887,-176.753,6.999,148.354
C04183=1207.188,279.759,-65.858,-176.755,6.997,148.354
C04184=1207.192,279.512,-65.830,-176.757,6.995,148.354
C04185=1207.196,279.263,-65.801,-176.760,6.992,148.354
C04186=1207.200,279.014,-65.773,-176.763,6.990,148.354
C04187=1207.205,278.766,-65.745,-176.765,6.987,148.354
C04188=1207.209,278.518,-65.717,-176.767,6.985,148.355
C04189=1207.214,278.270,-65.688,-176.771,6.982,148.355
C04190=1207.218,278.021,-65.660,-176.773,6.980,148.355
C04191=1207.223,277.773,-65.632,-176.775,6.977,148.355
C04192=1207.227,277.524,-65.604,-176.778,6.975,148.355
C04193=1207.232,277.276,-65.575,-176.780,6.973,148.355
C04194=1207.236,277.027,-65.547,-176.783,6.970,148.355
C04195=1207.241,276.779,-65.519,-176.785,6.968,148.355
C04196=1207.244,276.531,-65.491,-176.788,6.965,148.356
C04197=1207.249,276.283,-65.463,-176.790,6.963,148.356
C04198=1207.253,276.034,-65.434,-176.792,6.961,148.356
C04199=1207.258,275.786,-65.406,-176.796,6.958,148.356
C04200=1207.262,275.537,-65.378,-176.798,6.956,148.356
C04201=1207.266,275.289,-65.350,-176.800,6.953,148.356
C04202=1207.270,275.041,-65.322,-176.803,6.951,148.356
C04203=1207.275,274.793,-65.293,-176.806,6.948,148.356
C04204=1207.279,274.544,-65.265,-176.808,6.946,148.357
C04205=1207.283,274.296,-65.237,-176.811,6.944,148.357
C04206=1207.288,274.047,-65.209,-176.813,6.941,148.357
C04207=1207.292,273.799,-65.181,-176.815,6.939,148.357
C04208=1207.296,273.550,-65.153,-176.819,6.936,148.357
C04209=1207.301,273.302,-65.125,-176.821,6.934,148.357
C04210=1207.306,273.054,-65.097,-176.823,6.932,148.358
C04211=1207.309,272.805,-65.069,-176.826,6.929,148.358
C04212=1207.315,272.557,-65.041,-176.828,6.927,148.358
C04213=1207.319,272.308,-65.013,-176.831,6.924,148.358
C04214=1207.323,272.060,-64.985,-176.833,6.922,148.358
C04215=1207.327,271.811,-64.957,-176.836,6.920,148.358
C04216=1207.332,271.563,-64.930,-176.839,6.917,148.358
C04217=1207.336,271.315,-64.902,-176.841,6.915,148.358
C04218=1207.340,271.066,-64.874,-176.843,6.913,148.359
C04219=1207.345,270.818,-64.845,-176.846,6.910,148.359
C04220=1207.349,270.569,-64.818,-176.848,6.908,148.359
C04221=1207.354,270.321,-64.790,-176.851,6.905,148.359
C04222=1207.358,270.073,-64.762,-176.854,6.903,148.359
C04223=1207.363,269.824,-64.734,-176.856,6.901,148.359
C04224=1207.367,269.576,-64.707,-176.859,6.898,148.360
C04225=1207.372,269.328,-64.679,-176.861,6.896,148.360
C04226=1207.376,269.079,-64.651,-176.864,6.894,148.360
C04227=1207.380,268.831,-64.624,-176.866,6.891,148.360
C04228=1207.384,268.583,-64.596,-176.869,6.889,148.360
C04229=1207.389,268.334,-64.568,-176.872,6.886,148.360
C04230=1207.393,268.086,-64.540,-176.874,6.884,148.360
C04231=1207.398,267.837,-64.513,-176.876,6.882,148.361
C04232=1207.402,267.589,-64.485,-176.879,6.879,148.361
C04233=1207.406,267.340,-64.458,-176.881,6.877,148.361
C04234=1207.411,267.092,-64.430,-176.884,6.875,148.361
C04235=1207.416,266.843,-64.402,-176.887,6.872,148.361
C04236=1207.420,266.595,-64.374,-176.889,6.870,148.361
C04237=1207.425,266.346,-64.347,-176.891,6.868,148.361
C04238=1207.428,266.098,-64.319,-176.895,6.865,148.362
C04239=1207.433,265.849,-64.292,-176.897,6.863,148.362
C04240=1207.437,265.601,-64.264,-176.899,6.861,148.362
C04241=1207.441,265.352,-64.237,-176.902,6.858,148.362
C04242=1207.446,265.104,-64.209,-176.904,6.856,148.362
C04243=1207.450,264.856,-64.182,-176.907,6.853,148.363
C04244=1207.455,264.608,-64.154,-176.909,6.851,148.363
C04245=1207.459,264.359,-64.127,-176.912,6.849,148.363
C04246=1207.464,264.110,-64.100,-176.915,6.846,148.363
C04247=1207.468,263.862,-64.072,-176.917,6.844,148.363
C04248=1207.473,263.614,-64.045,-176.919,6.842,148.363
C04249=1207.477,263.341,-64.014,-176.923,6.839,148.364
C04250=1207.482,263.068,-63.984,-176.925,6.836,148.364
C04251=1207.487,262.796,-63.954,-176.928,6.834,148.364
C04252=1207.492,262.523,-63.924,-176.931,6.831,148.364
C04253=1207.496,262.274,-63.896,-176.933,6.830,148.364
C04254=1207.501,262.025,-63.869,-176.935,6.827,148.364
C04255=1207.505,261.777,-63.842,-176.939,6.825,148.365
C04256=1207.510,261.529,-63.814,-176.941,6.823,148.365
C04257=1207.514,261.280,-63.787,-176.943,6.821,148.365
C04258=1207.518,261.032,-63.761,-176.946,6.818,148.365
C04259=1207.522,260.784,-63.733,-176.949,6.816,148.365
C04260=1207.527,260.535,-63.706,-176.951,6.814,148.365
C04261=1207.532,260.287,-63.679,-176.954,6.811,148.366
C04262=1207.536,260.037,-63.651,-176.956,6.809,148.366
C04263=1207.540,259.789,-63.624,-176.959,6.807,148.366
C04264=1207.545,259.541,-63.596,-176.961,6.804,148.366
C04265=1207.549,259.293,-63.569,-176.964,6.802,148.366
C04266=1207.554,259.044,-63.542,-176.966,6.800,148.367
C04267=1207.559,258.796,-63.515,-176.969,6.797,148.367
C04268=1207.562,258.547,-63.488,-176.972,6.795,148.367
C04269=1207.567,258.298,-63.461,-176.974,6.793,148.367
C04270=1207.571,258.050,-63.434,-176.976,6.791,148.367
C04271=1207.576,257.802,-63.406,-176.979,6.788,148.368
C04272=1207.580,257.553,-63.379,-176.982,6.786,148.368
C04273=1207.585,257.305,-63.352,-176.984,6.784,148.368
C04274=1207.588,257.056,-63.326,-176.987,6.781,148.368
C04275=1207.593,256.807,-63.298,-176.990,6.779,148.368
C04276=1207.598,256.559,-63.271,-176.992,6.777,148.368
C04277=1207.602,256.310,-63.244,-176.994,6.775,148.369
C04278=1207.607,256.062,-63.217,-176.997,6.772,148.369
C04279=1207.611,255.814,-63.191,-177.000,6.770,148.369
C04280=1207.615,255.565,-63.164,-177.002,6.768,148.369
C04281=1207.620,255.317,-63.137,-177.005,6.765,148.369
C04282=1207.625,255.068,-63.110,-177.007,6.763,148.369
C04283=1207.629,254.820,-63.083,-177.010,6.761,148.370
C04284=1207.633,254.571,-63.056,-177.012,6.759,148.370
C04285=1207.637,254.322,-63.029,-177.015,6.757,148.370
C04286=1207.642,254.074,-63.002,-177.017,6.754,148.370
C04287=1207.646,253.826,-62.975,-177.020,6.753,148.371
C04288=1207.651,253.577,-62.949,-177.022,6.750,148.371
C04289=1207.656,253.328,-62.922,-177.025,6.748,148.371
C04290=1207.660,253.080,-62.895,-177.028,6.746,148.371
C04291=1207.664,252.831,-62.868,-177.030,6.744,148.371
C04292=1207.669,252.583,-62.841,-177.033,6.742,148.372
C04293=1207.673,252.334,-62.814,-177.035,6.739,148.372
C04294=1207.677,252.086,-62.788,-177.038,6.737,148.372
C04295=1207.682,251.837,-62.761,-177.040,6.735,148.372
C04296=1207.686,251.589,-62.735,-177.043,6.733,148.372
C04297=1207.691,251.341,-62.708,-177.045,6.730,148.372
C04298=1207.696,251.092,-62.681,-177.048,6.728,148.373
C04299=1207.700,250.844,-62.654,-177.051,6.726,148.373
C04300=1207.704,250.595,-62.628,-177.053,6.724,148.373
C04301=1207.709,250.346,-62.601,-177.056,6.721,148.373
C04302=1207.713,250.098,-62.574,-177.058,6.719,148.373
C04303=1207.718,249.850,-62.547,-177.061,6.717,148.374
C04304=1207.722,249.601,-62.522,-177.063,6.715,148.374
C04305=1207.727,249.352,-62.494,-177.066,6.712,148.374
C04306=1207.731,249.104,-62.467,-177.069,6.711,148.374
C04307=1207.735,248.855,-62.442,-177.071,6.708,148.375
C04308=1207.740,248.606,-62.415,-177.073,6.706,148.375
C04309=1207.744,248.358,-62.388,-177.076,6.703,148.375
C04310=1207.749,248.109,-62.362,-177.079,6.702,148.375
C04311=1207.753,247.861,-62.335,-177.081,6.700,148.376
C04312=1207.758,247.612,-62.308,-177.083,6.698,148.376
C04313=1207.762,247.364,-62.283,-177.086,6.696,148.376
C04314=1207.766,247.115,-62.255,-177.089,6.693,148.376
C04315=1207.771,246.866,-62.230,-177.091,6.691,148.376
C04316=1207.775,246.618,-62.203,-177.094,6.689,148.377
C04317=1207.780,246.369,-62.177,-177.096,6.687,148.377
C04318=1207.784,246.121,-62.150,-177.099,6.684,148.377
C04319=1207.788,245.872,-62.123,-177.102,6.682,148.377
C04320=1207.793,245.623,-62.097,-177.104,6.680,148.377
C04321=1207.797,245.375,-62.071,-177.107,6.678,148.378
C04322=1207.803,245.127,-62.045,-177.109,6.676,148.378
C04323=1207.807,244.878,-62.018,-177.112,6.673,148.378
C04324=1207.811,244.629,-61.992,-177.114,6.671,148.378
C04325=1207.815,244.381,-61.965,-177.117,6.669,148.378
C04326=1207.820,244.132,-61.940,-177.120,6.668,148.379
C04327=1207.825,243.883,-61.913,-177.122,6.665,148.379
C04328=1207.828,243.635,-61.887,-177.125,6.663,148.379
C04329=1207.833,243.386,-61.860,-177.127,6.661,148.379
C04330=1207.837,243.138,-61.834,-177.130,6.659,148.380
C04331=1207.842,242.890,-61.809,-177.132,6.657,148.380
C04332=1207.847,242.641,-61.781,-177.135,6.655,148.380
C04333=1207.851,242.392,-61.756,-177.138,6.652,148.380
C04334=1207.855,242.144,-61.730,-177.140,6.650,148.381
C04335=1207.860,241.895,-61.703,-177.142,6.648,148.381
C04336=1207.864,241.646,-61.677,-177.145,6.646,148.381
C04337=1207.869,241.397,-61.651,-177.148,6.644,148.381
C04338=1207.874,241.150,-61.625,-177.150,6.641,148.381
C04339=1207.878,240.901,-61.599,-177.153,6.639,148.382
C04340=1207.882,240.652,-61.573,-177.156,6.637,148.382
C04341=1207.887,240.404,-61.546,-177.158,6.635,148.382
C04342=1207.891,240.155,-61.520,-177.160,6.633,148.382
C04343=1207.895,239.906,-61.495,-177.163,6.632,148.383
C04344=1207.901,239.658,-61.469,-177.166,6.629,148.383
C04345=1207.905,239.409,-61.442,-177.168,6.627,148.383
C04346=1207.909,239.161,-61.416,-177.171,6.625,148.383
C04347=1207.913,238.912,-61.391,-177.173,6.623,148.384
C04348=1207.918,238.663,-61.364,-177.176,6.621,148.384
C04349=1207.923,238.415,-61.339,-177.178,6.619,148.384
C04350=1207.927,238.166,-61.312,-177.181,6.616,148.384
C04351=1207.931,237.918,-61.287,-177.184,6.614,148.385
C04352=1207.936,237.668,-61.260,-177.186,6.612,148.385
C04353=1207.941,237.397,-61.233,-177.189,6.610,148.385
C04354=1207.946,237.126,-61.204,-177.192,6.607,148.385
C04355=1207.950,236.854,-61.176,-177.194,6.606,148.386
C04356=1207.956,236.583,-61.148,-177.197,6.603,148.386
C04357=1207.960,236.335,-61.122,-177.200,6.601,148.386
C04358=1207.965,236.086,-61.095,-177.202,6.599,148.386
C04359=1207.969,235.837,-61.070,-177.205,6.597,148.387
C04360=1207.974,235.589,-61.044,-177.208,6.595,148.387
C04361=1207.978,235.340,-61.019,-177.210,6.593,148.387
C04362=1207.982,235.091,-60.993,-177.213,6.590,148.387
C04363=1207.987,234.843,-60.967,-177.216,6.588,148.388
C04364=1207.991,234.594,-60.942,-177.218,6.587,148.388
C04365=1207.996,234.345,-60.915,-177.220,6.584,148.388
C04366=1208.001,234.097,-60.890,-177.223,6.583,148.388
C04367=1208.005,233.848,-60.864,-177.226,6.581,148.389
C04368=1208.009,233.599,-60.838,-177.228,6.579,148.389
C04369=1208.014,233.350,-60.813,-177.231,6.576,148.389
C04370=1208.018,233.102,-60.787,-177.234,6.574,148.389
C04371=1208.023,232.854,-60.762,-177.236,6.572,148.390
C04372=1208.027,232.605,-60.736,-177.238,6.570,148.390
C04373=1208.032,232.357,-60.710,-177.241,6.568,148.390
C04374=1208.036,232.108,-60.685,-177.244,6.566,148.390
C04375=1208.040,231.858,-60.660,-177.246,6.565,148.391
C04376=1208.045,231.610,-60.634,-177.248,6.562,148.391
C04377=1208.050,231.362,-60.608,-177.252,6.560,148.391
C04378=1208.054,231.113,-60.583,-177.254,6.558,148.391
C04379=1208.059,230.864,-60.557,-177.257,6.556,148.392
C04380=1208.064,230.616,-60.531,-177.259,6.554,148.392
C04381=1208.068,230.367,-60.506,-177.262,6.552,148.392
C04382=1208.073,230.118,-60.481,-177.264,6.550,148.393
C04383=1208.076,229.869,-60.455,-177.267,6.548,148.393
C04384=1208.081,229.621,-60.430,-177.269,6.546,148.393
C04385=1208.085,229.373,-60.404,-177.272,6.543,148.393
C04386=1208.090,229.124,-60.379,-177.275,6.542,148.394
C04387=1208.095,228.875,-60.354,-177.277,6.540,148.394
C04388=1208.099,228.626,-60.328,-177.280,6.538,148.394
C04389=1208.104,228.378,-60.303,-177.282,6.536,148.394
C04390=1208.108,228.129,-60.277,-177.285,6.534,148.395
C04391=1208.113,227.880,-60.252,-177.288,6.532,148.395
C04392=1208.117,227.632,-60.227,-177.290,6.530,148.395
C04393=1208.122,227.383,-60.201,-177.292,6.528,148.395
C04394=1208.127,227.134,-60.176,-177.295,6.526,148.396
C04395=1208.131,226.885,-60.150,-177.298,6.523,148.396
C04396=1208.136,226.637,-60.125,-177.300,6.521,148.396
C04397=1208.140,226.388,-60.100,-177.303,6.519,148.396
C04398=1208.144,226.139,-60.075,-177.306,6.518,148.397
C04399=1208.149,225.891,-60.049,-177.308,6.516,148.397
C04400=1208.153,225.642,-60.024,-177.311,6.514,148.397
C04401=1208.158,225.394,-59.999,-177.313,6.512,148.398
C04402=1208.163,225.144,-59.974,-177.316,6.510,148.398
C04403=1208.167,224.896,-59.949,-177.318,6.508,148.398
C04404=1208.172,224.647,-59.923,-177.321,6.506,148.399
C04405=1208.176,224.399,-59.899,-177.324,6.504,148.399
C04406=1208.180,224.150,-59.873,-177.326,6.501,148.399
C04407=1208.185,223.902,-59.848,-177.329,6.500,148.399
C04408=1208.190,223.653,-59.823,-177.332,6.498,148.400
C04409=1208.195,223.404,-59.798,-177.334,6.496,148.400
C04410=1208.198,223.156,-59.773,-177.337,6.494,148.400
C04411=1208.203,222.907,-59.748,-177.339,6.492,148.400
C04412=1208.208,222.658,-59.722,-177.342,6.490,148.401
C04413=1208.213,222.409,-59.698,-177.344,6.488,148.401
C04414=1208.216,222.161,-59.673,-177.347,6.486,148.401
C04415=1208.221,221.912,-59.648,-177.350,6.484,148.402
C04416=1208.226,221.663,-59.623,-177.352,6.482,148.402
C04417=1208.231,221.415,-59.597,-177.354,6.480,148.402
C04418=1208.234,221.165,-59.573,-177.357,6.478,148.402
C04419=1208.239,220.917,-59.548,-177.360,6.476,148.403
C04420=1208.244,220.668,-59.523,-177.363,6.474,148.403
C04421=1208.248,220.419,-59.499,-177.365,6.472,148.403
C04422=1208.252,220.171,-59.473,-177.368,6.470,148.403
C04423=1208.258,219.922,-59.448,-177.370,6.468,148.404
C04424=1208.262,219.673,-59.422,-177.373,6.466,148.404
C04425=1208.266,219.425,-59.398,-177.375,6.465,148.404
C04426=1208.271,219.176,-59.374,-177.378,6.463,148.405
C04427=1208.276,218.927,-59.348,-177.381,6.461,148.405
C04428=1208.280,218.679,-59.324,-177.383,6.459,148.405
C04429=1208.284,218.429,-59.299,-177.386,6.457,148.406
C04430=1208.289,218.181,-59.275,-177.388,6.455,148.406
C04431=1208.294,217.933,-59.249,-177.391,6.453,148.406
C04432=1208.298,217.683,-59.224,-177.393,6.451,148.407
C04433=1208.303,217.435,-59.200,-177.396,6.450,148.407
C04434=1208.307,217.186,-59.175,-177.399,6.447,148.407
C04435=1208.311,216.938,-59.150,-177.401,6.445,148.407
C04436=1208.316,216.689,-59.126,-177.404,6.443,148.408
C04437=1208.321,216.440,-59.101,-177.407,6.441,148.408
C04438=1208.325,216.191,-59.077,-177.409,6.439,148.408
C04439=1208.330,215.942,-59.052,-177.412,6.437,148.409
C04440=1208.334,215.694,-59.027,-177.415,6.436,148.409
C04441=1208.339,215.445,-59.002,-177.417,6.434,148.409
C04442=1208.343,215.196,-58.978,-177.419,6.432,148.409
C04443=1208.348,214.947,-58.953,-177.422,6.430,148.410
C04444=1208.353,214.699,-58.928,-177.425,6.428,148.410
C04445=1208.357,214.450,-58.904,-177.427,6.426,148.410
C04446=1208.362,214.201,-58.879,-177.430,6.424,148.411
C04447=1208.366,213.952,-58.855,-177.433,6.422,148.411
C04448=1208.371,213.704,-58.829,-177.435,6.421,148.411
C04449=1208.375,213.455,-58.805,-177.438,6.419,148.412
C04450=1208.380,213.207,-58.781,-177.440,6.417,148.412
C04451=1208.384,212.957,-58.756,-177.443,6.415,148.412
C04452=1208.389,212.709,-58.731,-177.445,6.413,148.413
C04453=1208.393,212.460,-58.707,-177.448,6.411,148.413
C04454=1208.397,212.211,-58.683,-177.451,6.409,148.413
C04455=1208.402,211.962,-58.658,-177.453,6.407,148.414
C04456=1208.407,211.714,-58.634,-177.456,6.406,148.414
C04457=1208.412,211.444,-58.608,-177.459,6.403,148.414
C04458=1208.417,211.172,-58.581,-177.462,6.401,148.415
C04459=1208.422,210.902,-58.554,-177.464,6.399,148.415
C04460=1208.427,210.632,-58.528,-177.468,6.397,148.415
C04461=1208.432,210.384,-58.504,-177.470,6.395,148.415
C04462=1208.435,210.135,-58.479,-177.473,6.393,148.416
C04463=1208.440,209.886,-58.455,-177.476,6.391,148.416
C04464=1208.445,209.637,-58.431,-177.478,6.389,148.416
C04465=1208.450,209.388,-58.407,-177.481,6.387,148.417
C04466=1208.454,209.139,-58.382,-177.484,6.386,148.417
C04467=1208.458,208.891,-58.358,-177.486,6.383,148.417
C04468=1208.464,208.642,-58.333,-177.488,6.382,148.418
C04469=1208.468,208.393,-58.309,-177.491,6.380,148.418
C04470=1208.472,208.145,-58.285,-177.494,6.378,148.418
C04471=1208.477,207.895,-58.261,-177.496,6.376,148.419
C04472=1208.482,207.647,-58.237,-177.499,6.374,148.419
C04473=1208.486,207.398,-58.213,-177.502,6.372,148.419
C04474=1208.491,207.149,-58.188,-177.504,6.371,148.420
C04475=1208.495,206.900,-58.164,-177.507,6.369,148.420
C04476=1208.500,206.651,-58.140,-177.509,6.367,148.420
C04477=1208.505,206.402,-58.116,-177.512,6.365,148.421
C04478=1208.509,206.154,-58.092,-177.515,6.363,148.421
C04479=1208.514,205.906,-58.067,-177.517,6.361,148.421
C04480=1208.518,205.657,-58.044,-177.520,6.359,148.421
C04481=1208.523,205.407,-58.019,-177.522,6.358,148.422
C04482=1208.527,205.159,-57.995,-177.524,6.356,148.422
C04483=1208.532,204.910,-57.972,-177.527,6.355,148.423
C04484=1208.536,204.661,-57.948,-177.530,6.353,148.423
C04485=1208.541,204.413,-57.923,-177.532,6.351,148.423
C04486=1208.546,204.164,-57.900,-177.535,6.349,148.424
C04487=1208.550,203.914,-57.875,-177.538,6.347,148.424
C04488=1208.554,203.666,-57.851,-177.540,6.345,148.424
C04489=1208.559,203.417,-57.828,-177.543,6.344,148.425
C04490=1208.564,203.168,-57.803,-177.545,6.342,148.425
C04491=1208.569,202.919,-57.780,-177.548,6.340,148.425
C04492=1208.573,202.671,-57.756,-177.551,6.338,148.426
C04493=1208.578,202.422,-57.731,-177.553,6.336,148.426
C04494=1208.582,202.173,-57.708,-177.556,6.334,148.426
C04495=1208.586,201.924,-57.684,-177.559,6.333,148.427
C04496=1208.592,201.675,-57.660,-177.561,6.331,148.427
C04497=1208.596,201.427,-57.636,-177.564,6.329,148.427
C04498=1208.601,201.178,-57.612,-177.567,6.327,148.428
C04499=1208.605,200.929,-57.588,-177.569,6.325,148.428
C04500=1208.610,200.680,-57.565,-177.572,6.323,148.428
C04501=1208.614,200.432,-57.541,-177.575,6.322,148.429
C04502=1208.619,200.183,-57.517,-177.577,6.320,148.429
C04503=1208.623,199.934,-57.493,-177.579,6.318,148.429
C04504=1208.628,199.685,-57.470,-177.582,6.316,148.429
C04505=1208.632,199.436,-57.445,-177.585,6.314,148.430
C04506=1208.637,199.187,-57.422,-177.587,6.313,148.430
C04507=1208.642,198.938,-57.398,-177.589,6.311,148.431
C04508=1208.646,198.689,-57.374,-177.592,6.309,148.431
C04509=1208.651,198.440,-57.351,-177.595,6.307,148.431
C04510=1208.655,198.192,-57.327,-177.597,6.306,148.432
C04511=1208.660,197.943,-57.303,-177.600,6.304,148.432
C04512=1208.664,197.694,-57.279,-177.603,6.302,148.432
C04513=1208.669,197.445,-57.256,-177.605,6.300,148.433
C04514=1208.674,197.196,-57.233,-177.608,6.298,148.433
C04515=1208.678,196.948,-57.208,-177.611,6.297,148.433
C04516=1208.683,196.699,-57.185,-177.613,6.295,148.434
C04517=1208.688,196.450,-57.162,-177.616,6.293,148.434
C04518=1208.692,196.201,-57.138,-177.619,6.291,148.434
C04519=1208.697,195.952,-57.114,-177.621,6.290,148.435
C04520=1208.701,195.703,-57.091,-177.623,6.288,148.435
C04521=1208.706,195.454,-57.068,-177.626,6.286,148.435
C04522=1208.710,195.206,-57.044,-177.629,6.285,148.436
C04523=1208.715,194.957,-57.020,-177.631,6.283,148.436
C04524=1208.720,194.708,-56.997,-177.634,6.281,148.436
C04525=1208.725,194.459,-56.973,-177.637,6.279,148.437
C04526=1208.729,194.210,-56.949,-177.639,6.277,148.437
C04527=1208.733,193.962,-56.927,-177.642,6.275,148.437
C04528=1208.738,193.713,-56.903,-177.645,6.274,148.438
C04529=1208.742,193.464,-56.880,-177.647,6.272,148.438
C04530=1208.747,193.215,-56.857,-177.649,6.271,148.439
C04531=1208.752,192.966,-56.833,-177.652,6.269,148.439
C04532=1208.756,192.717,-56.809,-177.655,6.267,148.439
C04533=1208.761,192.468,-56.786,-177.658,6.266,148.440
C04534=1208.766,192.220,-56.763,-177.660,6.264,148.440
C04535=1208.771,191.971,-56.739,-177.663,6.262,148.441
C04536=1208.775,191.722,-56.717,-177.666,6.260,148.441
C04537=1208.780,191.473,-56.693,-177.668,6.258,148.441
C04538=1208.784,191.224,-56.670,-177.671,6.257,148.442
C04539=1208.789,190.975,-56.647,-177.673,6.256,148.442
C04540=1208.794,190.726,-56.623,-177.676,6.254,148.442
C04541=1208.798,190.478,-56.599,-177.678,6.252,148.443
C04542=1208.802,190.229,-56.576,-177.681,6.250,148.443
C04543=1208.807,189.980,-56.553,-177.684,6.248,148.443
C04544=1208.811,189.731,-56.530,-177.686,6.246,148.444
C04545=1208.817,189.482,-56.507,-177.689,6.245,148.444
C04546=1208.821,189.233,-56.483,-177.692,6.243,148.444
C04547=1208.825,188.985,-56.461,-177.694,6.242,148.445
C04548=1208.830,188.736,-56.437,-177.696,6.240,148.445
C04549=1208.835,188.487,-56.414,-177.699,6.238,148.445
C04550=1208.839,188.238,-56.390,-177.702,6.236,148.446
C04551=1208.844,187.988,-56.368,-177.704,6.235,148.446
C04552=1208.849,187.740,-56.345,-177.707,6.233,148.447
C04553=1208.854,187.491,-56.322,-177.710,6.231,148.447
C04554=1208.858,187.242,-56.299,-177.712,6.229,148.447
C04555=1208.862,186.993,-56.276,-177.714,6.228,148.448
C04556=1208.867,186.744,-56.253,-177.718,6.227,148.448
C04557=1208.872,186.495,-56.229,-177.720,6.225,148.449
C04558=1208.876,186.246,-56.206,-177.723,6.223,148.449
C04559=1208.881,185.998,-56.183,-177.726,6.221,148.449
C04560=1208.886,185.749,-56.160,-177.728,6.219,148.450
C04561=1208.890,185.479,-56.136,-177.731,6.218,148.450
C04562=1208.896,185.210,-56.111,-177.733,6.216,148.450
C04563=1208.901,184.940,-56.086,-177.737,6.214,148.451
C04564=1208.906,184.671,-56.061,-177.739,6.212,148.451
C04565=1208.910,184.421,-56.038,-177.742,6.211,148.452
C04566=1208.915,184.172,-56.015,-177.745,6.209,148.452
C04567=1208.919,183.923,-55.992,-177.747,6.208,148.452
C04568=1208.924,183.675,-55.969,-177.749,6.206,148.453
C04569=1208.928,183.426,-55.947,-177.752,6.204,148.453
C04570=1208.933,183.176,-55.924,-177.755,6.202,148.453
C04571=1208.938,182.927,-55.901,-177.757,6.200,148.454
C04572=1208.943,182.679,-55.878,-177.760,6.199,148.454
C04573=1208.947,182.430,-55.855,-177.763,6.198,148.455
C04574=1208.952,182.181,-55.833,-177.765,6.196,148.455
C04575=1208.956,181.932,-55.809,-177.768,6.194,148.455
C04576=1208.962,181.684,-55.786,-177.771,6.193,148.456
C04577=1208.966,181.434,-55.764,-177.773,6.191,148.456
C04578=1208.971,181.185,-55.741,-177.776,6.189,148.456
C04579=1208.975,180.937,-55.718,-177.778,6.188,148.457
C04580=1208.980,180.688,-55.696,-177.781,6.186,148.457
C04581=1208.984,180.439,-55.673,-177.783,6.184,148.458
C04582=1208.989,180.190,-55.650,-177.786,6.183,148.458
C04583=1208.993,179.940,-55.628,-177.789,6.181,148.458
C04584=1208.998,179.692,-55.605,-177.791,6.180,148.459
C04585=1209.003,179.443,-55.583,-177.794,6.178,148.459
C04586=1209.007,179.194,-55.559,-177.796,6.176,148.460
C04587=1209.012,178.945,-55.538,-177.799,6.175,148.460
C04588=1209.017,178.696,-55.514,-177.802,6.173,148.460
C04589=1209.021,178.447,-55.492,-177.804,6.172,148.461
C04590=1209.027,178.198,-55.469,-177.807,6.170,148.461
C04591=1209.031,177.950,-55.447,-177.809,6.168,148.461
C04592=1209.036,177.700,-55.424,-177.812,6.167,148.462
C04593=1209.039,177.451,-55.401,-177.815,6.165,148.462
C04594=1209.044,177.203,-55.380,-177.817,6.164,148.463
C04595=1209.049,176.954,-55.356,-177.820,6.162,148.463
C04596=1209.054,176.705,-55.334,-177.822,6.160,148.463
C04597=1209.059,176.456,-55.311,-177.825,6.158,148.464
C04598=1209.063,176.207,-55.289,-177.828,6.157,148.464
C04599=1209.068,175.958,-55.267,-177.830,6.156,148.465
C04600=1209.072,175.709,-55.244,-177.833,6.154,148.465
C04601=1209.077,175.460,-55.222,-177.836,6.152,148.465
C04602=1209.082,175.211,-55.199,-177.838,6.151,148.466
C04603=1209.086,174.962,-55.177,-177.840,6.150,148.466
C04604=1209.091,174.713,-55.155,-177.843,6.148,148.467
C04605=1209.096,174.464,-55.132,-177.846,6.146,148.467
C04606=1209.100,174.215,-55.110,-177.848,6.144,148.467
C04607=1209.105,173.967,-55.087,-177.852,6.143,148.468
C04608=1209.110,173.717,-55.065,-177.854,6.142,148.468
C04609=1209.114,173.468,-55.043,-177.856,6.140,148.469
C04610=1209.119,173.220,-55.020,-177.859,6.138,148.469
C04611=1209.124,172.970,-54.998,-177.862,6.136,148.469
C04612=1209.128,172.722,-54.976,-177.864,6.135,148.470
C04613=1209.133,172.472,-54.954,-177.866,6.133,148.470
C04614=1209.137,172.223,-54.931,-177.870,6.132,148.471
C04615=1209.142,171.975,-54.909,-177.872,6.130,148.471
C04616=1209.147,171.725,-54.887,-177.874,6.129,148.471
C04617=1209.152,171.476,-54.865,-177.877,6.127,148.472
C04618=1209.156,171.228,-54.842,-177.880,6.126,148.472
C04619=1209.161,170.979,-54.820,-177.882,6.124,148.473
C04620=1209.165,170.730,-54.798,-177.885,6.123,148.473
C04621=1209.171,170.481,-54.776,-177.888,6.121,148.474
C04622=1209.175,170.232,-54.753,-177.890,6.119,148.474
C04623=1209.180,169.983,-54.731,-177.893,6.118,148.474
C04624=1209.184,169.734,-54.709,-177.895,6.117,148.475
C04625=1209.189,169.484,-54.687,-177.898,6.115,148.475
C04626=1209.194,169.236,-54.665,-177.901,6.113,148.476
C04627=1209.198,168.986,-54.643,-177.903,6.112,148.476
C04628=1209.203,168.738,-54.621,-177.906,6.111,148.476
C04629=1209.207,168.489,-54.599,-177.908,6.109,148.477
C04630=1209.213,168.240,-54.576,-177.911,6.107,148.477
C04631=1209.217,167.991,-54.554,-177.914,6.105,148.477
C04632=1209.222,167.742,-54.533,-177.916,6.105,148.478
C04633=1209.226,167.493,-54.510,-177.919,6.103,148.478
C04634=1209.231,167.244,-54.489,-177.921,6.101,148.479
C04635=1209.235,166.995,-54.467,-177.924,6.100,148.479
C04636=1209.241,166.746,-54.444,-177.926,6.098,148.480
C04637=1209.245,166.496,-54.422,-177.929,6.097,148.480
C04638=1209.250,166.248,-54.401,-177.932,6.095,148.480
C04639=1209.255,165.999,-54.379,-177.934,6.094,148.481
C04640=1209.259,165.750,-54.357,-177.937,6.092,148.481
C04641=1209.264,165.501,-54.335,-177.939,6.090,148.482
C04642=1209.268,165.252,-54.313,-177.942,6.090,148.482
C04643=1209.273,165.003,-54.292,-177.945,6.088,148.483
C04644=1209.277,164.754,-54.270,-177.947,6.086,148.483
C04645=1209.283,164.505,-54.247,-177.950,6.084,148.483
C04646=1209.287,164.256,-54.225,-177.952,6.083,148.484
C04647=1209.292,164.007,-54.204,-177.955,6.082,148.484
C04648=1209.296,163.758,-54.181,-177.958,6.080,148.485
C04649=1209.301,163.509,-54.160,-177.960,6.079,148.485
C04650=1209.306,163.260,-54.138,-177.963,6.077,148.485
C04651=1209.310,163.011,-54.116,-177.965,6.075,148.486
C04652=1209.315,162.762,-54.094,-177.969,6.074,148.486
C04653=1209.320,162.512,-54.073,-177.971,6.073,148.487
C04654=1209.325,162.264,-54.051,-177.973,6.071,148.487
C04655=1209.329,162.015,-54.030,-177.976,6.069,148.487
C04656=1209.334,161.766,-54.008,-177.979,6.069,148.488
C04657=1209.339,161.517,-53.986,-177.981,6.067,148.488
C04658=1209.343,161.268,-53.964,-177.984,6.065,148.489
C04659=1209.348,161.019,-53.942,-177.986,6.064,148.489
C04660=1209.353,160.770,-53.921,-177.989,6.062,148.490
C04661=1209.357,160.520,-53.899,-177.992,6.061,148.490
C04662=1209.362,160.272,-53.878,-177.994,6.060,148.491
C04663=1209.367,160.023,-53.856,-177.997,6.058,148.491
C04664=1209.371,159.773,-53.835,-177.999,6.056,148.491
C04665=1209.376,159.505,-53.811,-178.002,6.055,148.492
C04666=1209.381,159.235,-53.788,-178.005,6.053,148.492
C04667=1209.386,158.966,-53.765,-178.008,6.052,148.493
C04668=1209.391,158.698,-53.741,-178.010,6.051,148.493
C04669=1209.396,158.448,-53.720,-178.013,6.049,148.494
C04670=1209.401,158.200,-53.698,-178.016,6.047,148.494
C04671=1209.406,157.950,-53.676,-178.018,6.046,148.495
C04672=1209.410,157.701,-53.656,-178.021,6.045,148.495
C04673=1209.415,157.453,-53.634,-178.024,6.043,148.495
C04674=1209.419,157.203,-53.612,-178.026,6.042,148.496
C04675=1209.424,156.954,-53.591,-178.029,6.040,148.496
C04676=1209.429,156.706,-53.569,-178.032,6.038,148.497
C04677=1209.433,156.456,-53.547,-178.034,6.038,148.497
C04678=1209.439,156.207,-53.526,-178.037,6.036,148.498
C04679=1209.443,155.959,-53.505,-178.039,6.034,148.498
C04680=1209.448,155.710,-53.484,-178.042,6.033,148.498
C04681=1209.452,155.460,-53.462,-178.044,6.031,148.499
C04682=1209.457,155.211,-53.441,-178.047,6.030,148.499
C04683=1209.462,154.962,-53.420,-178.050,6.029,148.500
C04684=1209.467,154.713,-53.398,-178.052,6.027,148.500
C04685=1209.471,154.464,-53.377,-178.054,6.026,148.501
C04686=1209.476,154.215,-53.356,-178.057,6.025,148.501
C04687=1209.481,153.966,-53.335,-178.060,6.023,148.502
C04688=1209.485,153.717,-53.313,-178.062,6.022,148.502
C04689=1209.490,153.467,-53.292,-178.065,6.021,148.503
C04690=1209.495,153.219,-53.270,-178.068,6.019,148.503
C04691=1209.500,152.970,-53.249,-178.070,6.018,148.503
C04692=1209.505,152.721,-53.228,-178.073,6.016,148.504
C04693=1209.509,152.471,-53.206,-178.076,6.015,148.504
C04694=1209.513,152.223,-53.185,-178.078,6.014,148.505
C04695=1209.519,151.974,-53.164,-178.081,6.012,148.505
C04696=1209.523,151.725,-53.143,-178.083,6.011,148.506
C04697=1209.528,151.475,-53.121,-178.086,6.009,148.506
C04698=1209.532,151.226,-53.101,-178.089,6.008,148.506
C04699=1209.537,150.977,-53.079,-178.091,6.007,148.507
C04700=1209.542,150.728,-53.058,-178.094,6.005,148.507
C04701=1209.547,150.480,-53.037,-178.097,6.003,148.508
C04702=1209.551,150.230,-53.016,-178.099,6.002,148.508
C04703=1209.556,149.981,-52.995,-178.102,6.001,148.509
C04704=1209.560,149.732,-52.974,-178.104,6.000,148.509
C04705=1209.566,149.483,-52.953,-178.107,5.998,148.510
C04706=1209.571,149.234,-52.932,-178.109,5.996,148.510
C04707=1209.575,148.985,-52.911,-178.112,5.996,148.511
C04708=1209.580,148.735,-52.890,-178.115,5.994,148.511
C04709=1209.585,148.486,-52.869,-178.117,5.993,148.511
C04710=1209.589,148.238,-52.848,-178.120,5.992,148.512
C04711=1209.594,147.989,-52.827,-178.123,5.990,148.512
C04712=1209.598,147.740,-52.806,-178.125,5.989,148.513
C04713=1209.604,147.490,-52.785,-178.128,5.987,148.513
C04714=1209.608,147.242,-52.764,-178.130,5.986,148.514
C04715=1209.612,146.992,-52.743,-178.133,5.985,148.514
C04716=1209.617,146.743,-52.722,-178.136,5.983,148.515
C04717=1209.622,146.494,-52.701,-178.138,5.982,148.515
C04718=1209.627,146.245,-52.680,-178.141,5.980,148.516
C04719=1209.632,145.996,-52.659,-178.143,5.979,148.516
C04720=1209.636,145.747,-52.638,-178.146,5.978,148.517
C04721=1209.642,145.498,-52.617,-178.149,5.976,148.517
C04722=1209.646,145.249,-52.597,-178.151,5.975,148.517
C04723=1209.650,144.999,-52.575,-178.154,5.974,148.518
C04724=1209.655,144.751,-52.555,-178.156,5.973,148.518
C04725=1209.660,144.501,-52.534,-178.159,5.971,148.519
C04726=1209.664,144.252,-52.513,-178.161,5.970,148.519
C04727=1209.670,144.003,-52.492,-178.164,5.969,148.520
C04728=1209.674,143.754,-52.472,-178.167,5.967,148.520
C04729=1209.679,143.505,-52.451,-178.169,5.966,148.521
C04730=1209.684,143.256,-52.431,-178.172,5.964,148.521
C04731=1209.688,143.007,-52.409,-178.174,5.963,148.521
C04732=1209.693,142.758,-52.389,-178.177,5.962,148.522
C04733=1209.698,142.509,-52.368,-178.179,5.961,148.522
C04734=1209.702,142.260,-52.347,-178.182,5.959,148.523
C04735=1209.708,142.011,-52.326,-178.185,5.958,148.523
C04736=1209.712,141.762,-52.306,-178.187,5.957,148.524
C04737=1209.717,141.512,-52.285,-178.190,5.955,148.524
C04738=1209.721,141.263,-52.264,-178.192,5.954,148.525
C04739=1209.726,141.014,-52.244,-178.195,5.953,148.525
C04740=1209.731,140.765,-52.223,-178.198,5.952,148.526
C04741=1209.735,140.516,-52.202,-178.200,5.950,148.526
C04742=1209.740,140.267,-52.182,-178.203,5.948,148.527
C04743=1209.745,140.018,-52.161,-178.206,5.948,148.527
C04744=1209.749,139.769,-52.141,-178.208,5.946,148.528
C04745=1209.754,139.519,-52.120,-178.210,5.945,148.528
C04746=1209.759,139.270,-52.099,-178.214,5.943,148.529
C04747=1209.764,139.021,-52.078,-178.216,5.943,148.529
C04748=1209.769,138.772,-52.059,-178.218,5.941,148.529
C04749=1209.773,138.523,-52.038,-178.221,5.940,148.530
C04750=1209.778,138.273,-52.017,-178.224,5.938,148.530
C04751=1209.783,138.024,-51.997,-178.226,5.937,148.531
C04752=1209.787,137.776,-51.977,-178.229,5.936,148.531
C04753=1209.792,137.526,-51.956,-178.232,5.934,148.532
C04754=1209.797,137.277,-51.935,-178.234,5.934,148.532
C04755=1209.802,137.029,-51.915,-178.237,5.932,148.533
C04756=1209.807,136.779,-51.895,-178.239,5.931,148.533
C04757=1209.812,136.530,-51.875,-178.242,5.929,148.534
C04758=1209.816,136.281,-51.854,-178.244,5.928,148.534
C04759=1209.821,136.032,-51.833,-178.247,5.927,148.535
C04760=1209.826,135.783,-51.813,-178.250,5.926,148.535
C04761=1209.831,135.534,-51.793,-178.252,5.924,148.536
C04762=1209.835,135.285,-51.773,-178.255,5.924,148.536
C04763=1209.840,135.035,-51.752,-178.258,5.922,148.537
C04764=1209.845,134.786,-51.732,-178.260,5.921,148.537
C04765=1209.849,134.537,-51.712,-178.263,5.919,148.538
C04766=1209.854,134.288,-51.692,-178.265,5.918,148.538
C04767=1209.859,134.039,-51.671,-178.268,5.917,148.539
C04768=1209.863,133.790,-51.650,-178.270,5.916,148.539
C04769=1209.869,133.521,-51.629,-178.273,5.915,148.540
C04770=1209.874,133.253,-51.607,-178.276,5.913,148.540
C04771=1209.879,132.984,-51.585,-178.279,5.912,148.541
C04772=1209.884,132.716,-51.563,-178.281,5.910,148.541
C04773=1209.889,132.466,-51.543,-178.285,5.909,148.542
C04774=1209.894,132.217,-51.523,-178.287,5.908,148.542
C04775=1209.899,131.967,-51.503,-178.289,5.906,148.543
C04776=1209.903,131.718,-51.483,-178.292,5.906,148.543
C04777=1209.908,131.470,-51.463,-178.295,5.904,148.544
C04778=1209.913,131.221,-51.443,-178.297,5.903,148.544
C04779=1209.918,130.971,-51.422,-178.300,5.901,148.545
C04780=1209.922,130.722,-51.402,-178.303,5.901,148.545
C04781=1209.927,130.473,-51.382,-178.305,5.899,148.546
C04782=1209.932,130.224,-51.362,-178.307,5.898,148.546
C04783=1209.936,129.974,-51.342,-178.311,5.897,148.547
C04784=1209.941,129.726,-51.322,-178.313,5.896,148.547
C04785=1209.946,129.476,-51.302,-178.316,5.894,148.548
C04786=1209.951,129.227,-51.281,-178.318,5.893,148.548
C04787=1209.956,128.978,-51.262,-178.321,5.891,148.548
C04788=1209.960,128.729,-51.241,-178.323,5.891,148.549
C04789=1209.965,128.479,-51.222,-178.326,5.889,148.549
C04790=1209.970,128.231,-51.202,-178.329,5.888,148.550
C04791=1209.975,127.981,-51.182,-178.331,5.887,148.551
C04792=1209.979,127.732,-51.162,-178.334,5.886,148.551
C04793=1209.984,127.483,-51.142,-178.336,5.885,148.552
C04794=1209.989,127.234,-51.122,-178.339,5.883,148.552
C04795=1209.994,126.985,-51.102,-178.341,5.883,148.553
C04796=1209.998,126.736,-51.082,-178.344,5.881,148.553
C04797=1210.003,126.486,-51.062,-178.347,5.880,148.554
C04798=1210.008,126.237,-51.042,-178.349,5.879,148.554
C04799=1210.012,125.988,-51.022,-178.352,5.878,148.555
C04800=1210.018,125.739,-51.003,-178.354,5.876,148.555
C04801=1210.022,125.490,-50.983,-178.357,5.875,148.555
C04802=1210.027,125.240,-50.963,-178.360,5.874,148.556
C04803=1210.031,124.992,-50.943,-178.362,5.873,148.556
C04804=1210.037,124.743,-50.923,-178.365,5.871,148.557
C04805=1210.041,124.493,-50.904,-178.367,5.870,148.557
C04806=1210.046,124.244,-50.883,-178.370,5.870,148.558
C04807=1210.051,123.995,-50.864,-178.372,5.868,148.558
C04808=1210.056,123.746,-50.844,-178.375,5.867,148.559
C04809=1210.060,123.497,-50.824,-178.378,5.866,148.560
C04810=1210.065,123.247,-50.804,-178.380,5.865,148.560
C04811=1210.070,122.998,-50.785,-178.383,5.863,148.561
C04812=1210.075,122.749,-50.765,-178.385,5.862,148.561
C04813=1210.080,122.500,-50.745,-178.388,5.861,148.562
C04814=1210.084,122.250,-50.725,-178.390,5.860,148.562
C04815=1210.090,122.001,-50.706,-178.393,5.859,148.563
C04816=1210.094,121.752,-50.686,-178.396,5.858,148.563
C04817=1210.099,121.503,-50.666,-178.398,5.857,148.564
C04818=1210.104,121.254,-50.647,-178.401,5.855,148.564
C04819=1210.108,121.005,-50.628,-178.404,5.855,148.565
C04820=1210.113,120.755,-50.608,-178.406,5.853,148.565
C04821=1210.118,120.507,-50.588,-178.409,5.852,148.566
C04822=1210.123,120.257,-50.568,-178.412,5.850,148.566
C04823=1210.127,120.008,-50.549,-178.414,5.849,148.567
C04824=1210.133,119.759,-50.529,-178.416,5.849,148.567
C04825=1210.138,119.509,-50.510,-178.419,5.847,148.568
C04826=1210.142,119.260,-50.489,-178.422,5.846,148.568
C04827=1210.147,119.012,-50.471,-178.424,5.845,148.569
C04828=1210.151,118.762,-50.451,-178.427,5.844,148.569
C04829=1210.156,118.513,-50.431,-178.430,5.842,148.570
C04830=1210.161,118.264,-50.412,-178.432,5.842,148.570
C04831=1210.166,118.014,-50.392,-178.434,5.841,148.571
C04832=1210.171,117.765,-50.373,-178.438,5.839,148.571
C04833=1210.176,117.516,-50.354,-178.440,5.838,148.572
C04834=1210.180,117.267,-50.334,-178.443,5.837,148.572
C04835=1210.185,117.017,-50.315,-178.445,5.836,148.573
C04836=1210.190,116.768,-50.295,-178.448,5.835,148.573
C04837=1210.194,116.520,-50.276,-178.450,5.834,148.574
C04838=1210.199,116.271,-50.256,-178.453,5.833,148.574
C04839=1210.204,116.021,-50.237,-178.456,5.831,148.575
C04840=1210.209,115.771,-50.217,-178.458,5.831,148.575
C04841=1210.214,115.523,-50.198,-178.460,5.830,148.576
C04842=1210.218,115.273,-50.179,-178.464,5.828,148.576
C04843=1210.224,115.025,-50.159,-178.466,5.827,148.577
C04844=1210.228,114.775,-50.140,-178.469,5.826,148.578
C04845=1210.232,114.526,-50.121,-178.471,5.825,148.578
C04846=1210.238,114.277,-50.101,-178.474,5.824,148.579
C04847=1210.243,114.027,-50.082,-178.476,5.823,148.579
C04848=1210.248,113.778,-50.063,-178.479,5.822,148.580
C04849=1210.252,113.528,-50.044,-178.482,5.820,148.580
C04850=1210.257,113.280,-50.025,-178.484,5.820,148.581
C04851=1210.262,113.030,-50.005,-178.486,5.819,148.581
C04852=1210.267,112.782,-49.987,-178.489,5.817,148.582
C04853=1210.272,112.532,-49.967,-178.492,5.816,148.582
C04854=1210.276,112.282,-49.947,-178.495,5.815,148.583
C04855=1210.281,112.034,-49.928,-178.497,5.814,148.583
C04856=1210.286,111.784,-49.909,-178.500,5.813,148.584
C04857=1210.291,111.535,-49.890,-178.502,5.812,148.584
C04858=1210.295,111.285,-49.871,-178.505,5.811,148.585
C04859=1210.301,111.037,-49.852,-178.507,5.810,148.585
C04860=1210.305,110.787,-49.832,-178.510,5.809,148.586
C04861=1210.310,110.539,-49.814,-178.512,5.808,148.586
C04862=1210.315,110.289,-49.794,-178.515,5.806,148.587
C04863=1210.320,110.040,-49.776,-178.518,5.805,148.587
C04864=1210.324,109.790,-49.756,-178.520,5.805,148.588
C04865=1210.330,109.541,-49.737,-178.523,5.803,148.588
C04866=1210.334,109.292,-49.718,-178.525,5.802,148.589
C04867=1210.339,109.043,-49.699,-178.528,5.801,148.589
C04868=1210.343,108.793,-49.680,-178.531,5.800,148.590
C04869=1210.349,108.544,-49.661,-178.533,5.799,148.591
C04870=1210.353,108.295,-49.642,-178.536,5.798,148.591
C04871=1210.358,108.046,-49.623,-178.539,5.797,148.592
C04872=1210.363,107.796,-49.604,-178.541,5.796,148.592
C04873=1210.368,107.529,-49.584,-178.544,5.795,148.593
C04874=1210.374,107.260,-49.564,-178.547,5.794,148.593
C04875=1210.379,106.991,-49.542,-178.549,5.792,148.594
C04876=1210.384,106.723,-49.522,-178.552,5.792,148.594
C04877=1210.388,106.473,-49.503,-178.555,5.790,148.595
C04878=1210.394,106.225,-49.484,-178.557,5.789,148.596
C04879=1210.398,105.975,-49.466,-178.560,5.789,148.596
C04880=1210.403,105.726,-49.446,-178.563,5.787,148.597
C04881=1210.407,105.477,-49.427,-178.565,5.786,148.597
C04882=1210.412,105.227,-49.409,-178.567,5.785,148.598
C04883=1210.418,104.979,-49.390,-178.570,5.784,148.598
C04884=1210.422,104.729,-49.371,-178.573,5.783,148.599
C04885=1210.427,104.480,-49.353,-178.575,5.782,148.599
C04886=1210.431,104.231,-49.333,-178.578,5.781,148.600
C04887=1210.437,103.981,-49.315,-178.581,5.780,148.600
C04888=1210.442,103.733,-49.296,-178.583,5.779,148.601
C04889=1210.447,103.482,-49.277,-178.586,5.778,148.601
C04890=1210.451,103.234,-49.259,-178.588,5.777,148.602
C04891=1210.456,102.984,-49.240,-178.591,5.776,148.602
C04892=1210.461,102.735,-49.221,-178.594,5.775,148.603
C04893=1210.466,102.486,-49.203,-178.596,5.774,148.604
C04894=1210.471,102.236,-49.183,-178.599,5.773,148.604
C04895=1210.475,101.987,-49.165,-178.602,5.772,148.605
C04896=1210.481,101.738,-49.146,-178.604,5.771,148.605
C04897=1210.485,101.488,-49.128,-178.606,5.770,148.606
C04898=1210.490,101.240,-49.109,-178.609,5.769,148.606
C04899=1210.495,100.990,-49.090,-178.612,5.768,148.607
C04900=1210.499,100.741,-49.071,-178.614,5.767,148.607
C04901=1210.504,100.492,-49.053,-178.617,5.766,148.608
C04902=1210.509,100.242,-49.034,-178.620,5.765,148.609
C04903=1210.514,99.993,-49.016,-178.622,5.764,148.609
C04904=1210.519,99.745,-48.997,-178.624,5.763,148.610
C04905=1210.524,99.494,-48.978,-178.627,5.762,148.610
C04906=1210.529,99.245,-48.960,-178.630,5.761,148.611
C04907=1210.533,98.997,-48.941,-178.632,5.760,148.611
C04908=1210.538,98.746,-48.922,-178.635,5.759,148.612
C04909=1210.543,98.497,-48.904,-178.638,5.758,148.612
C04910=1210.548,98.249,-48.886,-178.640,5.757,148.613
C04911=1210.553,97.999,-48.867,-178.643,5.756,148.614
C04912=1210.557,97.750,-48.848,-178.645,5.755,148.614
C04913=1210.562,97.501,-48.830,-178.648,5.754,148.615
C04914=1210.567,97.252,-48.812,-178.650,5.754,148.615
C04915=1210.572,97.001,-48.793,-178.653,5.752,148.616
C04916=1210.577,96.753,-48.775,-178.656,5.751,148.616
C04917=1210.582,96.504,-48.757,-178.658,5.750,148.617
C04918=1210.587,96.254,-48.738,-178.661,5.749,148.617
C04919=1210.591,96.005,-48.719,-178.663,5.748,148.618
C04920=1210.596,95.756,-48.701,-178.666,5.747,148.618
C04921=1210.601,95.507,-48.683,-178.668,5.747,148.619
C04922=1210.606,95.257,-48.665,-178.671,5.745,148.619
C04923=1210.611,95.008,-48.645,-178.674,5.745,148.620
C04924=1210.616,94.759,-48.627,-178.676,5.744,148.621
C04925=1210.621,94.510,-48.609,-178.679,5.742,148.621
C04926=1210.625,94.260,-48.591,-178.682,5.742,148.622
C04927=1210.631,94.010,-48.572,-178.684,5.741,148.622
C04928=1210.635,93.762,-48.554,-178.686,5.740,148.623
C04929=1210.640,93.512,-48.536,-178.689,5.738,148.623
C04930=1210.645,93.263,-48.517,-178.692,5.738,148.624
C04931=1210.649,93.013,-48.499,-178.694,5.737,148.625
C04932=1210.654,92.764,-48.481,-178.696,5.736,148.625
C04933=1210.660,92.515,-48.463,-178.700,5.735,148.626
C04934=1210.665,92.266,-48.444,-178.702,5.734,148.626
C04935=1210.669,92.016,-48.426,-178.704,5.733,148.627
C04936=1210.674,91.767,-48.408,-178.708,5.732,148.627
C04937=1210.679,91.518,-48.390,-178.710,5.731,148.628
C04938=1210.684,91.269,-48.372,-178.712,5.730,148.628
C04939=1210.689,91.020,-48.354,-178.715,5.730,148.629
C04940=1210.693,90.770,-48.336,-178.718,5.728,148.630
C04941=1210.699,90.520,-48.317,-178.720,5.727,148.630
C04942=1210.703,90.271,-48.299,-178.722,5.727,148.631
C04943=1210.708,90.022,-48.281,-178.725,5.726,148.631
C04944=1210.713,89.773,-48.263,-178.728,5.725,148.632
C04945=1210.718,89.524,-48.244,-178.730,5.724,148.632
C04946=1210.722,89.274,-48.226,-178.733,5.723,148.633
C04947=1210.727,89.025,-48.208,-178.736,5.722,148.634
C04948=1210.732,88.776,-48.190,-178.738,5.721,148.634
C04949=1210.737,88.527,-48.172,-178.741,5.720,148.635
C04950=1210.742,88.278,-48.154,-178.743,5.719,148.635
C04951=1210.747,88.028,-48.136,-178.746,5.719,148.636
C04952=1210.751,87.778,-48.119,-178.749,5.717,148.636
C04953=1210.756,87.529,-48.101,-178.751,5.716,148.637
C04954=1210.761,87.280,-48.083,-178.754,5.716,148.637
C04955=1210.766,87.030,-48.065,-178.756,5.715,148.638
C04956=1210.771,86.781,-48.047,-178.759,5.713,148.639
C04957=1210.776,86.532,-48.029,-178.762,5.713,148.639
C04958=1210.781,86.283,-48.011,-178.764,5.712,148.640
C04959=1210.786,86.034,-47.993,-178.766,5.711,148.640
C04960=1210.791,85.785,-47.975,-178.769,5.711,148.641
C04961=1210.795,85.535,-47.956,-178.772,5.709,148.641
C04962=1210.800,85.285,-47.938,-178.774,5.708,148.642
C04963=1210.805,85.036,-47.920,-178.777,5.708,148.643
C04964=1210.810,84.786,-47.903,-178.779,5.707,148.643
C04965=1210.815,84.537,-47.885,-178.782,5.705,148.644
C04966=1210.820,84.288,-47.867,-178.785,5.705,148.644
C04967=1210.825,84.039,-47.849,-178.787,5.704,148.645
C04968=1210.830,83.790,-47.831,-178.790,5.703,148.645
C04969=1210.835,83.541,-47.813,-178.792,5.703,148.646
C04970=1210.840,83.291,-47.796,-178.795,5.701,148.647
C04971=1210.845,83.042,-47.778,-178.798,5.700,148.647
C04972=1210.850,82.792,-47.760,-178.800,5.700,148.648
C04973=1210.854,82.543,-47.742,-178.802,5.699,148.648
C04974=1210.858,82.294,-47.724,-178.805,5.698,148.649
C04975=1210.863,82.044,-47.707,-178.808,5.697,148.650
C04976=1210.868,81.795,-47.689,-178.810,5.696,148.650
C04977=1210.873,81.526,-47.670,-178.813,5.696,148.651
C04978=1210.879,81.258,-47.651,-178.816,5.694,148.651
C04979=1210.884,80.990,-47.632,-178.819,5.694,148.652
C04980=1210.889,80.722,-47.612,-178.821,5.693,148.653
C04981=1210.895,80.472,-47.595,-178.824,5.691,148.653
C04982=1210.900,80.223,-47.577,-178.827,5.691,148.654
C04983=1210.904,79.974,-47.559,-178.829,5.690,148.654
C04984=1210.909,79.724,-47.543,-178.832,5.689,148.655
C04985=1210.914,79.475,-47.525,-178.834,5.689,148.655
C04986=1210.919,79.226,-47.507,-178.837,5.687,148.656
C04987=1210.924,78.976,-47.489,-178.839,5.686,148.657
C04988=1210.929,78.727,-47.471,-178.842,5.686,148.657
C04989=1210.934,78.478,-47.453,-178.845,5.685,148.658
C04990=1210.938,78.228,-47.437,-178.847,5.684,148.658
C04991=1210.943,77.979,-47.419,-178.850,5.683,148.659
C04992=1210.948,77.729,-47.401,-178.853,5.682,148.660
C04993=1210.953,77.480,-47.383,-178.855,5.681,148.660
C04994=1210.958,77.231,-47.366,-178.857,5.681,148.661
C04995=1210.963,76.981,-47.349,-178.860,5.680,148.661
C04996=1210.968,76.732,-47.331,-178.863,5.680,148.662
C04997=1210.973,76.482,-47.314,-178.865,5.678,148.662
C04998=1210.977,76.234,-47.296,-178.868,5.677,148.663
C04999=1210.982,75.984,-47.279,-178.871,5.677,148.664
C05000=1210.987,75.735,-47.261,-178.873,5.676,148.664
C05001=1210.992,75.485,-47.243,-178.875,5.675,148.665
C05002=1210.997,75.236,-47.226,-178.878,5.675,148.665
C05003=1211.001,74.987,-47.208,-178.881,5.673,148.666
C05004=1211.007,74.737,-47.191,-178.883,5.672,148.667
C05005=1211.011,74.489,-47.174,-178.886,5.672,148.667
C05006=1211.017,74.239,-47.157,-178.888,5.671,148.668
C05007=1211.022,73.990,-47.139,-178.891,5.670,148.668
C05008=1211.027,73.740,-47.122,-178.893,5.670,148.669
C05009=1211.031,73.491,-47.105,-178.896,5.668,148.669
C05010=1211.036,73.241,-47.087,-178.899,5.667,148.670
C05011=1211.041,72.992,-47.070,-178.901,5.667,148.671
C05012=1211.046,72.743,-47.052,-178.904,5.666,148.671
C05013=1211.051,72.493,-47.035,-178.906,5.665,148.672
C05014=1211.056,72.244,-47.017,-178.909,5.665,148.672
C05015=1211.061,71.995,-47.001,-178.912,5.663,148.673
C05016=1211.066,71.745,-46.983,-178.914,5.662,148.674
C05017=1211.070,71.496,-46.966,-178.917,5.662,148.674
C05018=1211.075,71.246,-46.949,-178.919,5.661,148.675
C05019=1211.080,70.997,-46.931,-178.922,5.660,148.675
C05020=1211.085,70.748,-46.914,-178.924,5.660,148.676
C05021=1211.090,70.498,-46.897,-178.927,5.659,148.677
C05022=1211.094,70.249,-46.879,-178.930,5.658,148.677
C05023=1211.100,70.000,-46.863,-178.932,5.657,148.678
C05024=1211.105,69.750,-46.845,-178.935,5.656,148.678
C05025=1211.109,69.501,-46.828,-178.937,5.656,148.679
C05026=1211.115,69.252,-46.811,-178.940,5.655,148.679
C05027=1211.119,69.002,-46.794,-178.942,5.654,148.680
C05028=1211.124,68.752,-46.777,-178.945,5.654,148.681
C05029=1211.129,68.504,-46.760,-178.948,5.652,148.681
C05030=1211.134,68.254,-46.742,-178.950,5.651,148.682
C05031=1211.140,68.005,-46.725,-178.953,5.651,148.682
C05032=1211.144,67.755,-46.709,-178.955,5.650,148.683
C05033=1211.149,67.506,-46.691,-178.958,5.649,148.684
C05034=1211.153,67.256,-46.674,-178.960,5.649,148.684
C05035=1211.159,67.007,-46.657,-178.963,5.648,148.685
C05036=1211.164,66.758,-46.640,-178.965,5.648,148.686
C05037=1211.169,66.509,-46.622,-178.968,5.646,148.686
C05038=1211.173,66.259,-46.606,-178.971,5.645,148.687
C05039=1211.178,66.009,-46.588,-178.973,5.645,148.687
C05040=1211.183,65.761,-46.572,-178.976,5.644,148.688
C05041=1211.189,65.511,-46.555,-178.978,5.643,148.688
C05042=1211.193,65.262,-46.537,-178.981,5.643,148.689
C05043=1211.198,65.012,-46.520,-178.983,5.642,148.690
C05044=1211.203,64.763,-46.504,-178.986,5.641,148.690
C05045=1211.208,64.514,-46.487,-178.989,5.640,148.691
C05046=1211.213,64.264,-46.470,-178.991,5.639,148.691
C05047=1211.217,64.015,-46.453,-178.994,5.639,148.692
C05048=1211.223,63.766,-46.436,-178.996,5.638,148.693
C05049=1211.228,63.516,-46.420,-178.999,5.637,148.693
C05050=1211.232,63.267,-46.402,-179.001,5.637,148.694
C05051=1211.237,63.017,-46.385,-179.004,5.636,148.695
C05052=1211.242,62.769,-46.369,-179.006,5.635,148.695
C05053=1211.247,62.519,-46.351,-179.009,5.635,148.696
C05054=1211.252,62.269,-46.335,-179.012,5.633,148.696
C05055=1211.257,62.020,-46.318,-179.015,5.633,148.697
C05056=1211.262,61.771,-46.301,-179.017,5.632,148.697
C05057=1211.267,61.521,-46.285,-179.019,5.631,148.698
C05058=1211.272,61.271,-46.267,-179.022,5.631,148.699
C05059=1211.276,61.022,-46.251,-179.025,5.630,148.699
C05060=1211.282,60.773,-46.234,-179.027,5.629,148.700
C05061=1211.287,60.523,-46.217,-179.030,5.629,148.701
C05062=1211.291,60.274,-46.200,-179.032,5.628,148.701
C05063=1211.297,60.025,-46.184,-179.035,5.628,148.702
C05064=1211.301,59.775,-46.167,-179.037,5.627,148.702
C05065=1211.306,59.526,-46.150,-179.040,5.625,148.703
C05066=1211.312,59.277,-46.133,-179.043,5.625,148.704
C05067=1211.316,59.027,-46.117,-179.045,5.624,148.704
C05068=1211.321,58.778,-46.100,-179.048,5.623,148.705
C05069=1211.326,58.529,-46.083,-179.050,5.623,148.705
C05070=1211.331,58.279,-46.066,-179.053,5.622,148.706
C05071=1211.336,58.029,-46.050,-179.055,5.622,148.707
C05072=1211.341,57.780,-46.034,-179.058,5.621,148.707
C05073=1211.346,57.531,-46.017,-179.060,5.620,148.708
C05074=1211.350,57.281,-46.000,-179.063,5.620,148.709
C05075=1211.356,57.032,-45.984,-179.065,5.619,148.709
C05076=1211.361,56.782,-45.967,-179.068,5.618,148.710
C05077=1211.365,56.533,-45.950,-179.071,5.617,148.710
C05078=1211.370,56.284,-45.934,-179.073,5.616,148.711
C05079=1211.375,56.034,-45.918,-179.076,5.616,148.712
C05080=1211.381,55.785,-45.901,-179.078,5.615,148.712
C05081=1211.386,55.516,-45.883,-179.081,5.614,148.713
C05082=1211.391,55.249,-45.865,-179.084,5.614,148.713
C05083=1211.396,54.979,-45.848,-179.086,5.613,148.714
C05084=1211.402,54.711,-45.829,-179.089,5.612,148.715
C05085=1211.406,54.462,-45.813,-179.092,5.611,148.715
C05086=1211.412,54.212,-45.797,-179.095,5.611,148.716
C05087=1211.416,53.963,-45.780,-179.097,5.610,148.717
C05088=1211.421,53.713,-45.763,-179.099,5.609,148.717
C05089=1211.426,53.464,-45.747,-179.102,5.609,148.718
C05090=1211.431,53.214,-45.731,-179.105,5.608,148.718
C05091=1211.436,52.965,-45.714,-179.107,5.608,148.719
C05092=1211.441,52.716,-45.698,-179.109,5.607,148.720
C05093=1211.446,52.467,-45.682,-179.112,5.606,148.720
C05094=1211.451,52.217,-45.665,-179.115,5.606,148.721
C05095=1211.456,51.967,-45.648,-179.117,5.605,148.722
C05096=1211.461,51.718,-45.632,-179.120,5.604,148.722
C05097=1211.466,51.468,-45.616,-179.122,5.604,148.723
C05098=1211.471,51.220,-45.600,-179.125,5.603,148.723
C05099=1211.475,50.970,-45.583,-179.127,5.602,148.724
C05100=1211.481,50.721,-45.567,-179.130,5.602,148.725
C05101=1211.485,50.471,-45.551,-179.132,5.601,148.725
C05102=1211.490,50.221,-45.534,-179.135,5.600,148.726
C05103=1211.496,49.972,-45.518,-179.138,5.599,148.726
C05104=1211.500,49.723,-45.501,-179.141,5.599,148.727
C05105=1211.505,49.474,-45.485,-179.143,5.598,148.728
C05106=1211.510,49.224,-45.469,-179.145,5.597,148.728
C05107=1211.515,48.975,-45.453,-179.148,5.597,148.729
C05108=1211.520,48.725,-45.437,-179.151,5.596,148.730
C05109=1211.525,48.476,-45.420,-179.153,5.595,148.730
C05110=1211.529,48.226,-45.404,-179.156,5.595,148.731
C05111=1211.535,47.977,-45.388,-179.158,5.594,148.731
C05112=1211.539,47.728,-45.372,-179.161,5.593,148.732
C05113=1211.545,47.478,-45.356,-179.163,5.593,148.733
C05114=1211.549,47.229,-45.339,-179.166,5.592,148.733
C05115=1211.555,46.979,-45.324,-179.169,5.592,148.734
C05116=1211.559,46.730,-45.307,-179.171,5.591,148.735
C05117=1211.564,46.480,-45.291,-179.174,5.590,148.735
C05118=1211.570,46.231,-45.274,-179.176,5.590,148.736
C05119=1211.575,45.981,-45.259,-179.179,5.589,148.737
C05120=1211.580,45.732,-45.242,-179.181,5.589,148.737
C05121=1211.585,45.482,-45.226,-179.184,5.588,148.738
C05122=1211.589,45.233,-45.210,-179.186,5.587,148.738
C05123=1211.594,44.984,-45.195,-179.189,5.587,148.739
C05124=1211.599,44.735,-45.178,-179.192,5.586,148.740
C05125=1211.604,44.485,-45.162,-179.194,5.586,148.740
C05126=1211.609,44.236,-45.146,-179.196,5.585,148.741
C05127=1211.614,43.986,-45.130,-179.199,5.584,148.741
C05128=1211.619,43.737,-45.115,-179.202,5.584,148.742
C05129=1211.624,43.487,-45.098,-179.204,5.583,148.743
C05130=1211.629,43.238,-45.082,-179.207,5.583,148.743
C05131=1211.634,42.988,-45.066,-179.209,5.582,148.744
C05132=1211.639,42.739,-45.050,-179.212,5.581,148.745
C05133=1211.644,42.489,-45.034,-179.214,5.581,148.745
C05134=1211.649,42.240,-45.018,-179.217,5.580,148.746
C05135=1211.654,41.991,-45.002,-179.220,5.579,148.747
C05136=1211.659,41.740,-44.986,-179.222,5.579,148.747
C05137=1211.664,41.492,-44.970,-179.224,5.578,148.748
C05138=1211.669,41.242,-44.954,-179.227,5.577,148.748
C05139=1211.673,40.992,-44.939,-179.230,5.577,148.749
C05140=1211.679,40.744,-44.923,-179.232,5.576,148.750
C05141=1211.683,40.494,-44.907,-179.234,5.576,148.750
C05142=1211.689,40.244,-44.891,-179.237,5.575,148.751
C05143=1211.694,39.995,-44.875,-179.240,5.574,148.752
C05144=1211.699,39.745,-44.859,-179.242,5.574,148.752
C05145=1211.704,39.496,-44.843,-179.245,5.573,148.753
C05146=1211.709,39.246,-44.828,-179.248,5.573,148.754
C05147=1211.713,38.997,-44.812,-179.250,5.572,148.754
C05148=1211.719,38.748,-44.796,-179.252,5.571,148.755
C05149=1211.723,38.498,-44.780,-179.255,5.571,148.755
C05150=1211.729,38.248,-44.765,-179.258,5.570,148.756
C05151=1211.734,38.000,-44.748,-179.260,5.570,148.757
C05152=1211.739,37.749,-44.732,-179.262,5.569,148.757
C05153=1211.743,37.500,-44.717,-179.265,5.568,148.758
C05154=1211.749,37.251,-44.702,-179.268,5.568,148.758
C05155=1211.753,37.002,-44.685,-179.270,5.567,148.759
C05156=1211.758,36.752,-44.669,-179.273,5.567,148.760
C05157=1211.764,36.503,-44.654,-179.276,5.566,148.760
C05158=1211.768,36.253,-44.638,-179.278,5.565,148.761
C05159=1211.773,36.004,-44.623,-179.280,5.565,148.762
C05160=1211.779,35.754,-44.607,-179.283,5.564,148.762
C05161=1211.783,35.504,-44.591,-179.286,5.564,148.763
C05162=1211.788,35.256,-44.576,-179.288,5.563,148.764
C05163=1211.793,35.006,-44.560,-179.291,5.563,148.764
C05164=1211.799,34.757,-44.544,-179.293,5.562,148.765
C05165=1211.803,34.507,-44.529,-179.296,5.561,148.765
C05166=1211.808,34.258,-44.514,-179.298,5.561,148.766
C05167=1211.813,34.008,-44.498,-179.301,5.560,148.767
C05168=1211.818,33.758,-44.482,-179.303,5.560,148.767
C05169=1211.824,33.509,-44.466,-179.306,5.560,148.768
C05170=1211.828,33.260,-44.451,-179.308,5.559,148.769
C05171=1211.834,33.010,-44.436,-179.311,5.558,148.769
C05172=1211.838,32.761,-44.419,-179.313,5.558,148.770
C05173=1211.843,32.512,-44.404,-179.316,5.557,148.771
C05174=1211.848,32.262,-44.389,-179.319,5.557,148.771
C05175=1211.853,32.012,-44.373,-179.321,5.556,148.772
C05176=1211.858,31.763,-44.358,-179.323,5.555,148.772
C05177=1211.863,31.514,-44.342,-179.326,5.555,148.773
C05178=1211.868,31.264,-44.326,-179.329,5.554,148.774
C05179=1211.872,31.014,-44.311,-179.331,5.554,148.774
C05180=1211.878,30.765,-44.296,-179.334,5.553,148.775
C05181=1211.883,30.516,-44.280,-179.337,5.553,148.776
C05182=1211.888,30.266,-44.265,-179.339,5.552,148.776
C05183=1211.893,30.017,-44.249,-179.341,5.551,148.777
C05184=1211.898,29.766,-44.234,-179.344,5.551,148.778
C05185=1211.903,29.498,-44.218,-179.347,5.550,148.778
C05186=1211.909,29.230,-44.201,-179.349,5.550,148.779
C05187=1211.915,28.961,-44.184,-179.352,5.549,148.780
C05188=1211.919,28.692,-44.168,-179.355,5.549,148.780
C05189=1211.925,28.443,-44.152,-179.357,5.548,148.781
C05190=1211.929,28.194,-44.137,-179.360,5.548,148.782
C05191=1211.934,27.944,-44.121,-179.363,5.547,148.782
C05192=1211.940,27.694,-44.107,-179.365,5.546,148.783
C05193=1211.944,27.445,-44.092,-179.368,5.546,148.784
C05194=1211.950,27.195,-44.076,-179.370,5.545,148.784
C05195=1211.955,26.946,-44.061,-179.373,5.545,148.785
C05196=1211.959,26.696,-44.045,-179.375,5.545,148.786
C05197=1211.964,26.447,-44.030,-179.377,5.544,148.786
C05198=1211.969,26.198,-44.014,-179.380,5.544,148.787
C05199=1211.974,25.948,-44.000,-179.383,5.543,148.788
C05200=1211.980,25.699,-43.985,-179.385,5.543,148.788
C05201=1211.984,25.449,-43.970,-179.388,5.542,148.789
C05202=1211.989,25.199,-43.954,-179.390,5.541,148.789
C05203=1211.995,24.950,-43.938,-179.393,5.541,148.790
C05204=1211.999,24.700,-43.924,-179.395,5.540,148.791
C05205=1212.005,24.451,-43.908,-179.398,5.540,148.791
C05206=1212.010,24.202,-43.893,-179.401,5.539,148.792
C05207=1212.015,23.952,-43.878,-179.403,5.539,148.793
C05208=1212.020,23.703,-43.863,-179.406,5.538,148.793
C05209=1212.024,23.453,-43.848,-179.408,5.538,148.794
C05210=1212.029,23.203,-43.832,-179.410,5.538,148.795
C05211=1212.034,22.954,-43.817,-179.413,5.537,148.795
C05212=1212.040,22.704,-43.802,-179.415,5.536,148.796
C05213=1212.044,22.455,-43.787,-179.418,5.536,148.797
C05214=1212.050,22.206,-43.772,-179.421,5.535,148.797
C05215=1212.054,21.957,-43.757,-179.423,5.535,148.798
C05216=1212.060,21.707,-43.742,-179.426,5.534,148.798
C05217=1212.065,21.458,-43.727,-179.428,5.533,148.799
C05218=1212.069,21.207,-43.711,-179.431,5.533,148.800
C05219=1212.074,20.958,-43.697,-179.433,5.533,148.800
C05220=1212.079,20.709,-43.682,-179.436,5.533,148.801
C05221=1212.085,20.459,-43.667,-179.438,5.532,148.802
C05222=1212.089,20.210,-43.652,-179.441,5.532,148.803
C05223=1212.095,19.960,-43.636,-179.443,5.531,148.803
C05224=1212.100,19.710,-43.622,-179.446,5.530,148.804
C05225=1212.104,19.461,-43.607,-179.448,5.530,148.804
C05226=1212.110,19.212,-43.592,-179.451,5.529,148.805
C05227=1212.115,18.962,-43.577,-179.454,5.529,148.806
C05228=1212.120,18.713,-43.562,-179.456,5.528,148.806
C05229=1212.125,18.463,-43.547,-179.458,5.528,148.807
C05230=1212.130,18.214,-43.532,-179.461,5.528,148.808
C05231=1212.135,17.964,-43.518,-179.463,5.527,148.808
C05232=1212.140,17.715,-43.503,-179.466,5.527,148.809
C05233=1212.144,17.465,-43.487,-179.468,5.526,148.810
C05234=1212.150,17.215,-43.472,-179.471,5.525,148.810
C05235=1212.154,16.966,-43.457,-179.474,5.525,148.811
C05236=1212.159,16.716,-43.443,-179.476,5.524,148.812
C05237=1212.165,16.467,-43.427,-179.478,5.525,148.812
C05238=1212.170,16.217,-43.413,-179.481,5.524,148.813
C05239=1212.174,15.968,-43.398,-179.483,5.523,148.813
C05240=1212.180,15.718,-43.383,-179.486,5.523,148.814
C05241=1212.185,15.469,-43.368,-179.489,5.522,148.815
C05242=1212.190,15.219,-43.354,-179.491,5.522,148.815
C05243=1212.194,14.970,-43.339,-179.494,5.521,148.816
C05244=1212.200,14.720,-43.324,-179.497,5.521,148.817
C05245=1212.205,14.471,-43.309,-179.499,5.520,148.818
C05246=1212.210,14.221,-43.295,-179.501,5.521,148.818
C05247=1212.215,13.972,-43.281,-179.503,5.520,148.819
C05248=1212.220,13.722,-43.265,-179.506,5.519,148.819
C05249=1212.225,13.473,-43.251,-179.509,5.519,148.820
C05250=1212.230,13.223,-43.236,-179.511,5.518,148.821
C05251=1212.235,12.974,-43.221,-179.514,5.518,148.821
C05252=1212.240,12.724,-43.207,-179.517,5.517,148.822
C05253=1212.245,12.475,-43.192,-179.519,5.517,148.823
C05254=1212.250,12.226,-43.178,-179.521,5.517,148.823
C05255=1212.255,11.977,-43.163,-179.524,5.516,148.824
C05256=1212.261,11.727,-43.148,-179.526,5.515,148.825
C05257=1212.266,11.477,-43.134,-179.529,5.515,148.825
C05258=1212.270,11.228,-43.119,-179.531,5.514,148.826
C05259=1212.275,10.978,-43.104,-179.534,5.514,148.827
C05260=1212.280,10.728,-43.090,-179.536,5.514,148.827
C05261=1212.286,10.479,-43.074,-179.539,5.514,148.828
C05262=1212.291,10.229,-43.060,-179.541,5.513,148.829
C05263=1212.296,9.979,-43.046,-179.544,5.513,148.829
C05264=1212.300,9.730,-43.031,-179.547,5.512,148.830
C05265=1212.305,9.481,-43.017,-179.549,5.511,148.831
C05266=1212.310,9.231,-43.002,-179.552,5.511,148.831
C05267=1212.316,8.981,-42.987,-179.554,5.511,148.832
C05268=1212.320,8.732,-42.972,-179.556,5.511,148.833
C05269=1212.326,8.483,-42.959,-179.559,5.510,148.833
C05270=1212.331,8.233,-42.944,-179.562,5.509,148.834
C05271=1212.336,7.983,-42.930,-179.564,5.509,148.835
C05272=1212.341,7.734,-42.915,-179.567,5.508,148.835
C05273=1212.346,7.485,-42.901,-179.569,5.509,148.836
C05274=1212.350,7.235,-42.886,-179.571,5.508,148.836
C05275=1212.356,6.985,-42.872,-179.574,5.507,148.837
C05276=1212.361,6.736,-42.857,-179.576,5.507,148.838
C05277=1212.366,6.486,-42.842,-179.579,5.506,148.839
C05278=1212.371,6.237,-42.828,-179.582,5.506,148.839
C05279=1212.376,5.987,-42.814,-179.584,5.505,148.840
C05280=1212.381,5.738,-42.800,-179.586,5.506,148.841
C05281=1212.386,5.488,-42.786,-179.589,5.505,148.841
C05282=1212.391,5.239,-42.771,-179.592,5.505,148.842
C05283=1212.396,4.989,-42.756,-179.594,5.504,148.843
C05284=1212.401,4.739,-42.742,-179.597,5.503,148.843
C05285=1212.406,4.490,-42.728,-179.599,5.503,148.844
C05286=1212.411,4.241,-42.714,-179.601,5.503,148.844
C05287=1212.416,3.991,-42.700,-179.604,5.502,148.845
C05288=1212.421,3.741,-42.685,-179.607,5.502,148.846
C05289=1212.426,3.472,-42.670,-179.609,5.501,148.847
C05290=1212.432,3.203,-42.654,-179.612,5.501,148.847
C05291=1212.438,2.934,-42.638,-179.615,5.500,148.848
C05292=1212.444,2.665,-42.624,-179.618,5.500,148.849
C05293=1212.448,2.416,-42.609,-179.620,5.499,148.849
C05294=1212.453,2.166,-42.594,-179.622,5.500,148.850
C05295=1212.458,1.917,-42.580,-179.625,5.499,148.851
C05296=1212.463,1.667,-42.566,-179.627,5.499,148.851
C05297=1212.469,1.418,-42.552,-179.630,5.498,148.852
C05298=1212.474,1.168,-42.538,-179.633,5.498,148.853
C05299=1212.479,0.919,-42.523,-179.635,5.497,148.853
C05300=1212.484,0.669,-42.509,-179.637,5.497,148.854
C05301=1212.489,0.419,-42.495,-179.640,5.497,148.855
C05302=1212.494,0.170,-42.481,-179.643,5.496,148.856
C05303=1212.499,-0.080,-42.467,-179.645,5.496,148.856
C05304=1212.503,-0.329,-42.453,-179.647,5.495,148.857
C05305=1212.508,-0.579,-42.439,-179.650,5.495,148.857
C05306=1212.514,-0.828,-42.425,-179.652,5.495,148.858
C05307=1212.519,-1.077,-42.410,-179.655,5.494,148.859
C05308=1212.524,-1.327,-42.396,-179.657,5.494,148.859
C05309=1212.529,-1.577,-42.383,-179.660,5.493,148.860
C05310=1212.534,-1.827,-42.368,-179.662,5.494,148.861
C05311=1212.539,-2.076,-42.354,-179.665,5.493,148.861
C05312=1212.544,-2.326,-42.340,-179.668,5.493,148.862
C05313=1212.549,-2.576,-42.326,-179.670,5.492,148.863
C05314=1212.555,-2.825,-42.312,-179.672,5.491,148.863
C05315=1212.559,-3.074,-42.298,-179.674,5.492,148.864
C05316=1212.564,-3.324,-42.284,-179.677,5.491,148.865
C05317=1212.569,-3.573,-42.270,-179.680,5.491,148.865
C05318=1212.575,-3.822,-42.256,-179.682,5.490,148.866
C05319=1212.580,-4.073,-42.242,-179.685,5.490,148.867
C05320=1212.585,-4.322,-42.228,-179.687,5.490,148.867
C05321=1212.590,-4.572,-42.214,-179.690,5.489,148.868
C05322=1212.595,-4.821,-42.200,-179.692,5.489,148.869
C05323=1212.600,-5.071,-42.186,-179.695,5.488,148.870
C05324=1212.605,-5.320,-42.172,-179.698,5.488,148.870
C05325=1212.610,-5.570,-42.159,-179.699,5.488,148.871
C05326=1212.615,-5.820,-42.144,-179.702,5.487,148.871
C05327=1212.620,-6.069,-42.130,-179.705,5.487,148.872
C05328=1212.625,-6.318,-42.117,-179.707,5.486,148.873
C05329=1212.630,-6.568,-42.102,-179.710,5.486,148.873
C05330=1212.635,-6.818,-42.089,-179.712,5.486,148.874
C05331=1212.641,-7.067,-42.075,-179.715,5.486,148.875
C05332=1212.646,-7.317,-42.061,-179.717,5.485,148.876
C05333=1212.650,-7.566,-42.047,-179.720,5.485,148.876
C05334=1212.655,-7.816,-42.033,-179.722,5.485,148.877
C05335=1212.661,-8.065,-42.020,-179.725,5.484,148.878
C05336=1212.666,-8.315,-42.005,-179.727,5.484,148.878
C05337=1212.671,-8.564,-41.992,-179.730,5.483,148.879
C05338=1212.676,-8.814,-41.978,-179.732,5.483,148.879
C05339=1212.681,-9.064,-41.964,-179.734,5.483,148.880
C05340=1212.686,-9.313,-41.950,-179.737,5.482,148.881
C05341=1212.691,-9.563,-41.937,-179.740,5.482,148.882
C05342=1212.696,-9.813,-41.923,-179.742,5.481,148.882
C05343=1212.701,-10.062,-41.909,-179.744,5.482,148.883
C05344=1212.706,-10.312,-41.896,-179.747,5.481,148.884
C05345=1212.711,-10.561,-41.882,-179.750,5.481,148.884
C05346=1212.716,-10.810,-41.868,-179.752,5.480,148.885
C05347=1212.722,-11.061,-41.854,-179.754,5.481,148.886
C05348=1212.727,-11.309,-41.841,-179.756,5.480,148.886
C05349=1212.731,-11.559,-41.827,-179.759,5.479,148.887
C05350=1212.737,-11.810,-41.813,-179.762,5.479,148.888
C05351=1212.742,-12.058,-41.800,-179.764,5.478,148.888
C05352=1212.747,-12.309,-41.786,-179.767,5.478,148.889
C05353=1212.752,-12.558,-41.772,-179.769,5.478,148.890
C05354=1212.757,-12.807,-41.759,-179.772,5.477,148.890
C05355=1212.762,-13.057,-41.745,-179.775,5.477,148.891
C05356=1212.767,-13.306,-41.731,-179.777,5.477,148.892
C05357=1212.772,-13.556,-41.718,-179.779,5.477,148.892
C05358=1212.778,-13.805,-41.704,-179.782,5.476,148.893
C05359=1212.783,-14.056,-41.691,-179.785,5.476,148.894
C05360=1212.787,-14.305,-41.677,-179.787,5.476,148.894
C05361=1212.793,-14.554,-41.663,-179.789,5.475,148.895
C05362=1212.797,-14.804,-41.650,-179.791,5.475,148.896
C05363=1212.803,-15.053,-41.636,-179.794,5.474,148.896
C05364=1212.808,-15.303,-41.623,-179.796,5.475,148.897
C05365=1212.813,-15.552,-41.609,-179.799,5.474,148.898
C05366=1212.818,-15.802,-41.596,-179.802,5.474,148.898
C05367=1212.823,-16.051,-41.583,-179.804,5.473,148.899
C05368=1212.828,-16.301,-41.569,-179.806,5.473,148.900
C05369=1212.833,-16.552,-41.555,-179.809,5.473,148.900
C05370=1212.838,-16.800,-41.542,-179.812,5.472,148.901
C05371=1212.843,-17.051,-41.529,-179.814,5.472,148.902
C05372=1212.848,-17.300,-41.515,-179.816,5.472,148.903
C05373=1212.853,-17.550,-41.502,-179.818,5.471,148.903
C05374=1212.858,-17.799,-41.488,-179.821,5.471,148.904
C05375=1212.864,-18.049,-41.475,-179.824,5.470,148.904
C05376=1212.869,-18.298,-41.461,-179.826,5.471,148.905
C05377=1212.874,-18.548,-41.448,-179.829,5.470,148.906
C05378=1212.879,-18.798,-41.435,-179.831,5.470,148.906
C05379=1212.884,-19.047,-41.421,-179.833,5.470,148.907
C05380=1212.890,-19.297,-41.408,-179.836,5.470,148.908
C05381=1212.894,-19.546,-41.394,-179.839,5.469,148.909
C05382=1212.900,-19.796,-41.381,-179.841,5.469,148.909
C05383=1212.904,-20.046,-41.368,-179.843,5.469,148.910
C05384=1212.910,-20.295,-41.354,-179.846,5.468,148.911
C05385=1212.914,-20.545,-41.341,-179.849,5.468,148.911
C05386=1212.920,-20.794,-41.328,-179.851,5.467,148.912
C05387=1212.924,-21.044,-41.314,-179.853,5.467,148.912
C05388=1212.930,-21.293,-41.301,-179.856,5.467,148.913
C05389=1212.935,-21.543,-41.288,-179.858,5.466,148.914
C05390=1212.940,-21.792,-41.274,-179.861,5.466,148.915
C05391=1212.945,-22.042,-41.262,-179.863,5.466,148.915
C05392=1212.951,-22.292,-41.248,-179.866,5.466,148.916
C05393=1212.955,-22.561,-41.234,-179.868,5.465,148.917
C05394=1212.962,-22.830,-41.220,-179.871,5.465,148.917
C05395=1212.967,-23.100,-41.205,-179.874,5.465,148.918
C05396=1212.972,-23.370,-41.191,-179.876,5.465,148.919
C05397=1212.978,-23.619,-41.178,-179.879,5.465,148.920
C05398=1212.982,-23.869,-41.164,-179.881,5.464,148.920
C05399=1212.987,-24.118,-41.152,-179.884,5.463,148.921
C05400=1212.993,-24.368,-41.138,-179.886,5.463,148.922
C05401=1212.998,-24.618,-41.125,-179.888,5.463,148.922
C05402=1213.004,-24.867,-41.112,-179.891,5.463,148.923
C05403=1213.008,-25.117,-41.099,-179.893,5.463,148.924
C05404=1213.013,-25.366,-41.086,-179.896,5.462,148.924
C05405=1213.018,-25.616,-41.072,-179.898,5.462,148.925
C05406=1213.023,-25.866,-41.060,-179.901,5.461,148.926
C05407=1213.028,-26.115,-41.047,-179.903,5.462,148.926
C05408=1213.033,-26.365,-41.033,-179.906,5.461,148.927
C05409=1213.038,-26.614,-41.020,-179.908,5.461,148.928
C05410=1213.044,-26.864,-41.007,-179.911,5.461,148.929
C05411=1213.049,-27.114,-40.994,-179.913,5.461,148.929
C05412=1213.054,-27.363,-40.982,-179.916,5.460,148.930
C05413=1213.059,-27.613,-40.968,-179.918,5.459,148.930
C05414=1213.064,-27.862,-40.955,-179.920,5.460,148.931
C05415=1213.069,-28.111,-40.942,-179.923,5.459,148.932
C05416=1213.074,-28.362,-40.929,-179.925,5.459,148.932
C05417=1213.080,-28.611,-40.916,-179.928,5.459,148.933
C05418=1213.084,-28.861,-40.903,-179.930,5.458,148.934
C05419=1213.090,-29.110,-40.890,-179.933,5.458,148.935
C05420=1213.095,-29.360,-40.877,-179.935,5.458,148.935
C05421=1213.100,-29.610,-40.864,-179.938,5.458,148.936
C05422=1213.105,-29.859,-40.852,-179.940,5.457,148.937
C05423=1213.111,-30.109,-40.838,-179.943,5.457,148.937
C05424=1213.115,-30.359,-40.825,-179.945,5.457,148.938
C05425=1213.120,-30.608,-40.813,-179.948,5.457,148.939
C05426=1213.126,-30.858,-40.800,-179.950,5.456,148.939
C05427=1213.131,-31.108,-40.787,-179.952,5.456,148.940
C05428=1213.136,-31.357,-40.774,-179.955,5.456,148.941
C05429=1213.141,-31.606,-40.761,-179.957,5.455,148.941
C05430=1213.146,-31.857,-40.748,-179.959,5.456,148.942
C05431=1213.151,-32.106,-40.735,-179.962,5.455,148.943
C05432=1213.156,-32.355,-40.723,-179.965,5.455,148.943
C05433=1213.161,-32.605,-40.710,-179.967,5.455,148.944
C05434=1213.167,-32.855,-40.697,-179.969,5.454,148.945
C05435=1213.172,-33.104,-40.684,-179.972,5.454,148.945
C05436=1213.177,-33.354,-40.671,-179.974,5.454,148.946
C05437=1213.182,-33.604,-40.658,-179.977,5.454,148.947
C05438=1213.187,-33.853,-40.646,-179.979,5.453,148.948
C05439=1213.193,-34.103,-40.633,-179.982,5.453,148.948
C05440=1213.197,-34.353,-40.620,-179.984,5.453,148.949
C05441=1213.202,-34.602,-40.607,-179.986,5.452,148.949
C05442=1213.207,-34.851,-40.594,-179.989,5.452,148.950
C05443=1213.212,-35.101,-40.582,-179.991,5.452,148.951
C05444=1213.218,-35.351,-40.568,-179.994,5.452,148.952
C05445=1213.223,-35.600,-40.556,-179.996,5.451,148.952
C05446=1213.228,-35.850,-40.543,-179.999,5.452,148.953
C05447=1213.233,-36.100,-40.531,179.999,5.451,148.954
C05448=1213.238,-36.349,-40.518,179.996,5.451,148.954
C05449=1213.243,-36.599,-40.506,179.994,5.451,148.955
C05450=1213.249,-36.848,-40.492,179.991,5.450,148.956
C05451=1213.253,-37.098,-40.479,179.989,5.450,148.956
C05452=1213.259,-37.348,-40.467,179.987,5.450,148.957
C05453=1213.264,-37.597,-40.454,179.984,5.450,148.958
C05454=1213.269,-37.847,-40.442,179.982,5.449,148.958
C05455=1213.274,-38.096,-40.430,179.980,5.449,148.959
C05456=1213.279,-38.346,-40.417,179.977,5.449,148.960
C05457=1213.284,-38.596,-40.404,179.974,5.448,148.960
C05458=1213.290,-38.845,-40.391,179.972,5.449,148.961
C05459=1213.295,-39.095,-40.379,179.970,5.448,148.962
C05460=1213.300,-39.345,-40.366,179.967,5.448,148.963
C05461=1213.305,-39.595,-40.354,179.965,5.448,148.963
C05462=1213.310,-39.844,-40.341,179.962,5.448,148.964
C05463=1213.315,-40.094,-40.329,179.960,5.447,148.965
C05464=1213.320,-40.343,-40.316,179.958,5.447,148.965
C05465=1213.325,-40.593,-40.303,179.955,5.447,148.966
C05466=1213.330,-40.842,-40.291,179.952,5.447,148.967
C05467=1213.336,-41.092,-40.279,179.950,5.447,148.967
C05468=1213.341,-41.342,-40.266,179.948,5.446,148.968
C05469=1213.346,-41.591,-40.254,179.945,5.446,148.969
C05470=1213.351,-41.840,-40.241,179.943,5.446,148.969
C05471=1213.356,-42.091,-40.229,179.941,5.445,148.970
C05472=1213.361,-42.340,-40.216,179.938,5.445,148.971
C05473=1213.366,-42.590,-40.204,179.936,5.445,148.971
C05474=1213.371,-42.840,-40.192,179.933,5.445,148.972
C05475=1213.377,-43.089,-40.179,179.931,5.445,148.973
C05476=1213.382,-43.338,-40.167,179.928,5.445,148.974
C05477=1213.386,-43.589,-40.154,179.926,5.444,148.974
C05478=1213.392,-43.838,-40.142,179.924,5.445,148.975
C05479=1213.397,-44.087,-40.129,179.921,5.444,148.976
C05480=1213.402,-44.337,-40.117,179.918,5.444,148.976
